(* Logix 5000 project; controller VET 1756-L62 rev 19.52; software revision 19.01; part 3 of 27 *)

        [202].S.BITS1.8   // 100-TOR-010 Atollo
        [586].S.BITS1.9   // 120-CAN-011 Conf. Cerrado
        [562].S.BITS1.9   // 110-TDC-004/2 Sobrecarga
        [318].S.BITS1.0   // 80-FIL-001 Enable
        [318].S.BITS1.1   // 80-FIL-001 Falla Resumen
        [318].S.BITS1.2   // 80-FIL-001 Conf Pos Abrir
        [318].S.BITS1.4   // 80-FIL-001 Conf Pos Cerrar
        [318].S.BITS1.26   // 80-FIL-001FLL
        [318].S.BITS1.27   // 80-FIL-001FV0
        [318].S.BITS1.28   // 80-FIL-001FATO
        [318].S.BITS1.29   // 80-FIL-001 Falla Abrir
        [318].S.BITS1.30   // 80-FIL-001 Falla Cerrar
        [318].S.BITS2.20   // 80-FIL-001 Reset Falla
        [318].S.BITS2.23   // 80-FIL-001 Test
        [318].S.BITS2.27   // 80-FIL-001 Cmd. Open
        [318].S.BITS2.30   // 80-FIL-001 OUT CLOSE
        [318].S.BITS2.31   // 80-FIL-001 OUT OPEN
        [319].S.BITS1.0   // 80-VEN-001 Enable
        [319].S.BITS1.1   // 80-VEN-001 Falla Resumen
        [319].S.BITS1.2   // 80-VEN-001 Conf. Marcha
        [319].S.BITS1.4   // 80-VEN-001 Cmd. Automatico
        [319].S.BITS1.26   // 80-VEN-001 FLL
        [319].S.BITS1.27   // 80-VEN-001 FV0
        [319].S.BITS1.28   // 80-VEN-001 FATO
        [319].S.BITS1.30   // 80-VEN-001 Falla Partida
        [319].S.BITS2.20   // 80-VEN-001 Reset Falla
        [319].S.BITS2.23   // 80-VEN-001 Test
        [319].S.BITS2.27   // 80-VEN-001 Cmd. Marcha
        [319].S.BITS2.30   // 80-VEN-001 OUT MARCHA
        [320].S.BITS1.0   // 8-VRT-638 Enable
        [320].S.BITS1.1   // 8-VRT-638 Falla Resumen
        [320].S.BITS1.2   // 8-VRT-638 Conf. Marcha
        [320].S.BITS1.4   // 8-VRT-638 Cmd. Automatico
        [320].S.BITS1.26   // 8-VRT-638 FLL
        [320].S.BITS1.27   // 8-VRT-638 FV0
        [320].S.BITS1.28   // 8-VRT-638 FATO
        [320].S.BITS1.30   // 8-VRT-638 Falla Partida
        [320].S.BITS2.20   // 8-VRT-638 Reset Falla
        [320].S.BITS2.23   // 8-VRT-638 Test
        [320].S.BITS2.27   // 8-VRT-638 Cmd. Marcha
        [320].S.BITS2.30   // 8-VRT-638 OUT MARCHA
        [322].S.BITS1.7   // 80-ENH-001 LLL
        [323].S.BITS1.0   // 8-ENF-630-2 Enable
        [323].S.BITS1.1   // 8-ENF-630-2 Falla Resumen
        [323].S.BITS1.2   // 8-ENF-630-2 Conf. Marcha
        [323].S.BITS1.4   // 8-ENF-630-2 Cmd. Automatico
        [323].S.BITS1.26   // 8-ENF-630-2 FLL
        [323].S.BITS1.27   // 8-ENF-630-2 FV0
        [323].S.BITS1.28   // 8-ENF-630-2 FATO
        [323].S.BITS1.30   // 8-ENF-630-2 Falla Partida
        [323].S.BITS2.20   // 8-ENF-630-2 Reset Falla
        [323].S.BITS2.23   // 8-ENF-630-2 Test
        [323].S.BITS2.27   // 8-ENF-630-2 Cmd. Marcha
        [323].S.BITS2.30   // 8-ENF-630-2 OUT MARCHA
        [324].S.BITS1.8   // L4-TOLV-002-B1 LL
        [235].S.BITS1.0   // 7-LRT-1189 Enable
        [325].S.BITS1.0   // 8-ENF-640-1 Enable
        [325].S.BITS1.1   // 8-ENF-640-1 Falla Resumen
        [325].S.BITS1.2   // 8-ENF-640-1 Conf. Marcha
        [325].S.BITS1.4   // 8-ENF-640-1 Cmd. Automatico
        [236].S.BITS1.0   // 100-CAN-025 Enable
        [325].S.BITS1.26   // 8-ENF-640-1 FLL
        [325].S.BITS1.27   // 8-ENF-640-1 FV0
        [325].S.BITS1.28   // 8-ENF-640-1 FATO
        [325].S.BITS1.30   // 8-ENF-640-1 Falla Partida
        [325].S.BITS2.20   // 8-ENF-640-1 Reset Falla
        [325].S.BITS2.23   // 8-ENF-640-1 Test
        [325].S.BITS2.27   // 8-ENF-640-1 Cmd. Marcha
        [325].S.BITS2.30   // 8-ENF-640-1 OUT MARCHA
        [326].S.BITS1.0   // 100-ELV-003 Enable
        [326].S.BITS1.1   // 100-ELV-003 Falla Resumen
        [326].S.BITS1.2   // 100-ELV-003 Conf. Marcha
        [326].S.BITS1.4   // 100-ELV-003 Cmd. Automatico
        [326].S.BITS1.26   // 100-ELV-003 FLL
        [326].S.BITS1.27   // 100-ELV-003 FV0
        [326].S.BITS1.28   // 100-ELV-003 FATO
        [326].S.BITS1.30   // 100-ELV-003 Falla Partida
        [326].S.BITS2.20   // 100-ELV-003 Reset Falla
        [326].S.BITS2.23   // 100-ELV-003 Test
        [326].S.BITS2.27   // 100-ELV-003 Cmd. Marcha
        [326].S.BITS2.30   // 100-ELV-003 OUT MARCHA
        [327].S.BITS1.26   // 8-ENF-640-2 FLL
        [327].S.BITS1.27   // 8-ENF-640-2 FV0
        [327].S.BITS1.28   // 8-ENF-640-2 FATO
        [328].S.BITS1.0   // 80-ESC-002/5 Enable
        [328].S.BITS1.1   // 80-ESC-002/5 Falla Resumen
        [328].S.BITS1.2   // 80-ESC-002/5 Conf. Marcha
        [328].S.BITS1.4   // 80-ESC-002/5 Cmd. Automatico
        [328].S.BITS1.26   // 80-ESC-002/5 FLL
        [328].S.BITS1.27   // 80-ESC-002/5 FV0
        [328].S.BITS1.28   // 80-ESC-002/5 FATO
        [328].S.BITS1.30   // 80-ESC-002/5 Falla Partida
        [328].S.BITS2.20   // 80-ESC-002/5 Reset Falla
        [328].S.BITS2.23   // 80-ESC-002/5 Test
        [328].S.BITS2.27   // 80-ESC-002/5 Cmd. Marcha
        [328].S.BITS2.30   // 80-ESC-002/5 OUT MARCHA
        [329].S.BITS1.0   // 80-VEN-002/5 Enable
        [329].S.BITS1.1   // 80-VEN-002/5 Falla Resumen
        [329].S.BITS1.2   // 80-VEN-002/5 Conf. Marcha
        [329].S.BITS1.4   // 80-VEN-002/5 Cmd. Automatico
        [329].S.BITS1.26   // 80-VEN-002/5 FLL
        [329].S.BITS1.27   // 80-VEN-002/5 FV0
        [329].S.BITS1.28   // 80-VEN-002/5 FATO
        [329].S.BITS1.30   // 80-VEN-002/5 Falla Partida
        [329].S.BITS2.20   // 80-VEN-002/5 Reset Falla
        [329].S.BITS2.23   // 80-VEN-002/5 Test
        [329].S.BITS2.27   // 80-VEN-002/5 Cmd. Marcha
        [329].S.BITS2.30   // 80-VEN-002/5 OUT MARCHA
        [331].S.BITS1.0   // 80-TOR-004/5 Enable
        [331].S.BITS1.1   // 80-TOR-004/5 Falla Resumen
        [331].S.BITS1.2   // 80-TOR-004/5 Conf. Marcha
        [331].S.BITS1.4   // 80-TOR-004/5 Cmd. Automatico
        [331].S.BITS1.26   // 80-TOR-004/5 FLL
        [331].S.BITS1.27   // 80-TOR-004/5 FV0
        [331].S.BITS1.28   // 80-TOR-004/5 FATO
        [331].S.BITS1.30   // 80-TOR-004/5 Falla Partida
        [331].S.BITS2.20   // 80-TOR-004/5 Reset Falla
        [331].S.BITS2.23   // 80-TOR-004/5 Test
        [331].S.BITS2.27   // 80-TOR-004/5 Cmd. Marcha
        [331].S.BITS2.30   // 80-TOR-004/5 OUT MARCHA
        [332].S.BITS1.0   // 8-VEN-647 Enable
        [332].S.BITS1.1   // 8-VEN-647 Falla Resumen
        [332].S.BITS1.2   // 8-VEN-647 Conf. Marcha
        [332].S.BITS1.4   // 8-VEN-647 Cmd. Automatico
        [332].S.BITS1.26   // 8-VEN-647 FLL
        [332].S.BITS1.27   // 8-VEN-647 FV0
        [332].S.BITS1.28   // 8-VEN-647 FATO
        [332].S.BITS1.30   // 8-VEN-647 Falla Partida
        [332].S.BITS2.20   // 8-VEN-647 Reset Falla
        [332].S.BITS2.23   // 8-VEN-647 Test
        [332].S.BITS2.27   // 8-VEN-647 Cmd. Marcha
        [332].S.BITS2.30   // 8-VEN-647 OUT MARCHA
        [333].S.BITS1.0   // 8-ENF-640-2 Enable
        [333].S.BITS1.1   // 8-ENF-640-2 Falla Resumen
        [333].S.BITS1.2   // 8-ENF-640-2 Conf. Marcha
        [333].S.BITS1.4   // 8-ENF-640-2 Cmd. Automatico
        [333].S.BITS1.26   // 8-ENF-640-2 FLL
        [333].S.BITS1.27   // 8-ENF-640-2 FV0
        [333].S.BITS1.28   // 8-ENF-640-2 FATO
        [333].S.BITS1.30   // 8-ENF-640-2 Falla Partida
        [333].S.BITS2.20   // 8-ENF-640-2 Reset Falla
        [333].S.BITS2.23   // 8-ENF-640-2 Test
        [333].S.BITS2.27   // 8-ENF-640-2 Cmd. Marcha
        [333].S.BITS2.30   // 8-ENF-640-2 OUT MARCHA
        [564].S.BITS1.9   // 110-ELV-001/2 Sobrecarga
        [236].S.BITS2.30   // 100-CAN-025 OUT CLOSE
        [355].S.BITS1.10   // 110-CAN-003 Conf. Abierto
        [587].S.BITS1.9   // 120-CAN-012 Conf. Cerrado
        [239].S.BITS2.31   // 7-CON-1192 OUT OPEN
        [242].S.BITS2.31   // 7-CON-1195 OUT OPEN
        [280].S.BITS1.8   // 100-DOS-100-M10 Atollo
        [335].S.BITS1.0   // 8-ROS-654 Enable
        [335].S.BITS1.1   // 8-ROS-654 Falla Resumen
        [335].S.BITS1.2   // 8-ROS-654 Conf. Marcha
        [335].S.BITS1.4   // 8-ROS-654 Cmd. Automatico
        [335].S.BITS1.26   // 8-ROS-654 FLL
        [335].S.BITS1.27   // 8-ROS-654 FV0
        [335].S.BITS1.28   // 8-ROS-654 FATO
        [335].S.BITS1.30   // 8-ROS-654 Falla Partida
        [335].S.BITS2.20   // 8-ROS-654 Reset Falla
        [335].S.BITS2.23   // 8-ROS-654 Test
        [335].S.BITS2.27   // 8-ROS-654 Cmd. Marcha
        [335].S.BITS2.30   // 8-ROS-654 OUT MARCHA
        [336].S.BITS1.0   // 8-ELV-656 Enable
        [336].S.BITS1.1   // 8-ELV-656 Falla Resumen
        [336].S.BITS1.2   // 8-ELV-656 Conf. Marcha
        [336].S.BITS1.4   // 8-ELV-656 Cmd. Automatico
        [336].S.BITS1.26   // 8-ELV-656 FLL
        [336].S.BITS1.27   // 8-ELV-656 FV0
        [336].S.BITS1.28   // 8-ELV-656 FATO
        [336].S.BITS1.30   // 8-ELV-656 Falla Partida
        [336].S.BITS2.20   // 8-ELV-656 Reset Falla
        [336].S.BITS2.23   // 8-ELV-656 Test
        [336].S.BITS2.27   // 8-ELV-656 Cmd. Marcha
        [336].S.BITS2.30   // 8-ELV-656 OUT MARCHA
        [565].S.BITS1.9   // 120-TDC-001/2 Sobrecarga
        [244].S.BITS2.31   // 100-TOR-020 OUT MARCHA
        [356].S.BITS1.10   // 110-CAN-004 Conf. Abierto
        [588].S.BITS1.9   // 120-CAN-013 Conf. Cerrado
        [246].S.BITS2.31   // 100-TOR-019 OUT MARCHA
        [248].S.BITS2.31   // 100-TOR-018 OUT MARCHA
        [282].S.BITS1.8   // 100-DOS-100-M11 Atollo
        [338].S.BITS1.0   // 8-RED-660 Enable
        [338].S.BITS1.1   // 8-RED-660 Falla Resumen
        [338].S.BITS1.2   // 8-RED-660 Conf. Marcha
        [338].S.BITS1.4   // 8-RED-660 Cmd. Automatico
        [338].S.BITS1.7   // TOLV-008 LLL
        [338].S.BITS1.8   // TOLV-008 LL
        [338].S.BITS1.9   // TOLV-008 LM
        [338].S.BITS1.10   // TOLV-008 LH
        [338].S.BITS1.26   // 8-RED-660 FLL
        [338].S.BITS1.27   // 8-RED-660 FV0
        [338].S.BITS1.28   // 8-RED-660 FATO
        [338].S.BITS1.30   // 8-RED-660 Falla Partida
        [338].S.BITS2.20   // 8-RED-660 Reset Falla
        [338].S.BITS2.23   // 8-RED-660 Test
        [338].S.BITS2.27   // 8-RED-660 Cmd. Marcha
        [338].S.BITS2.30   // 8-RED-660 OUT MARCHA
        [339].S.BITS1.0   // 8-ELV-662 Enable
        [339].S.BITS1.1   // 8-ELV-662 Falla Resumen
        [339].S.BITS1.2   // 8-ELV-662 Conf. Marcha
        [339].S.BITS1.4   // 8-ELV-662 Cmd. Automatico
        [339].S.BITS1.26   // 8-ELV-662 FLL
        [339].S.BITS1.27   // 8-ELV-662 FV0
        [339].S.BITS1.28   // 8-ELV-662 FATO
        [339].S.BITS1.29   // CV-ENF-L1 Falla Abrir
        [339].S.BITS2.20   // 8-ELV-662 Reset Falla
        [339].S.BITS2.23   // 8-ELV-662 Test
        [339].S.BITS2.31   // CV-ENF-L1 OUT OPEN
        [340].S.BITS1.0   // 8-ZRD-664 Enable
        [340].S.BITS1.1   // 8-ZRD-664 Falla Resumen
        [340].S.BITS1.2   // 8-ZRD-664 Conf. Marcha
        [340].S.BITS1.4   // 8-ZRD-664 Cmd. Automatico
        [340].S.BITS1.7   // 80-TOL-004/6 LLL
        [340].S.BITS1.8   // 80-TOL-004/6 LL
        [340].S.BITS1.9   // 80-TOL-004/6 LM
        [340].S.BITS1.10   // 80-TOL-004/6 LH
        [340].S.BITS1.26   // 8-ZRD-664 FLL
        [340].S.BITS1.27   // 8-ZRD-664 FV0
        [340].S.BITS1.28   // 8-ZRD-664 FATO
        [340].S.BITS1.30   // 8-ZRD-664 Falla Partida
        [340].S.BITS2.20   // 8-ZRD-664 Reset Falla
        [340].S.BITS2.23   // 8-ZRD-664 Test
        [340].S.BITS2.27   // 8-ZRD-664 Cmd. Marcha
        [340].S.BITS2.30   // 8-ZRD-664 OUT MARCHA
        [341].S.BITS1.0   // 8-RED-666 Enable
        [341].S.BITS1.1   // 8-RED-666 Falla Resumen
        [341].S.BITS1.2   // 8-RED-666 Conf. Marcha
        [341].S.BITS1.4   // 8-RED-666 Cmd. Automatico
        [341].S.BITS1.26   // 8-RED-666 FLL
        [341].S.BITS1.27   // 8-RED-666 FV0
        [341].S.BITS1.28   // 8-RED-666 FATO
        [341].S.BITS1.30   // 8-RED-666 Falla Partida
        [341].S.BITS2.20   // 8-RED-666 Reset Falla
        [341].S.BITS2.23   // 8-RED-666 Test
        [341].S.BITS2.27   // 8-RED-666 Cmd. Marcha
        [341].S.BITS2.30   // 8-RED-666 OUT MARCHA
        [342].S.BITS1.0   // 8-CON-664b Enable
        [342].S.BITS1.1   // 8-CON-664b Falla Resumen
        [342].S.BITS1.4   // 8-CON-664b Conf Pos Cerrar
        [342].S.BITS1.26   // 110-TDC-001 FLL
        [342].S.BITS1.27   // 110-TDC-001 FV0
        [342].S.BITS1.28   // 110-TDC-001 FATO
        [342].S.BITS1.30   // 8-CON-664b Falla Cerrar
        [342].S.BITS2.20   // 8-CON-664b Reset Falla
        [342].S.BITS2.23   // 8-CON-664b Test
        [342].S.BITS2.27   // 8-CON-664b Cmd. Open
        [342].S.BITS2.30   // 8-CON-664b OUT CLOSE
        [343].S.BITS1.0   // COM-VIR-1 Enable
        [343].S.BITS1.1   // COM-VIR-1 Falla Resumen
        [343].S.BITS1.2   // COM-VIR-1 Conf Pos Abrir
        [343].S.BITS1.4   // COM-VIR-1 Conf Pos Cerrar
        [343].S.BITS1.29   // COM-VIR-1 Falla Abrir
        [343].S.BITS1.30   // COM-VIR-1 Falla Cerrar
        [343].S.BITS2.20   // COM-VIR-1 Reset Falla
        [343].S.BITS2.23   // COM-VIR-1 Test
        [343].S.BITS2.27   // COM-VIR-1 Cmd. Open
        [343].S.BITS2.30   // COM-VIR-1 OUT CLOSE
        [343].S.BITS2.31   // COM-VIR-1 OUT OPEN
        [337].S.BITS1.8   // 110-VEN-003 Atollo
        [357].S.BITS1.10   // 110-CAN-005 Conf. Abierto
        [589].S.BITS1.9   // 120-CAN-014 Conf. Cerrado
        [169].S.BITS1.10   // 100-VEN-002 Velocidad Cero
        [344].S.BITS1.26   // 80-EXP-002/6 FLL
        [344].S.BITS1.27   // 80-EXP-002/6 FV0
        [344].S.BITS1.28   // 80-EXP-002/6 FATO
        [116].S.BITS1.10   // 100-ELV-001 Velocidad Cero
        [590].S.BITS1.9   // 120-CAN-015 Conf. Cerrado
        [205].S.BITS1.8   // 100-TOR-036 Atollo
        [344].S.BITS2.27   // 110-LMG-001-01 Cmd. Open
        [571].S.BITS1.9   // 110-TDC-003/3 Sobrecarga
        [345].S.BITS1.0   // 80-DES-002/6 Enable
        [345].S.BITS1.1   // 80-DES-002/6 Falla Resumen
        [345].S.BITS1.2   // 80-DES-002/6 Conf. Marcha
        [345].S.BITS1.4   // 80-DES-002/6 Cmd. Automatico
        [345].S.BITS1.26   // 80-DES-002/6 FLL
        [345].S.BITS1.27   // 80-DES-002/6 FV0
        [345].S.BITS1.28   // 80-DES-002/6 FATO
        [345].S.BITS1.30   // 80-DES-002/6 Falla Partida
        [345].S.BITS2.20   // 80-DES-002/6 Reset Falla
        [345].S.BITS2.23   // 80-DES-002/6 Test
        [345].S.BITS2.27   // 80-DES-002/6 Cmd. Marcha
        [345].S.BITS2.30   // 80-DES-002/6 OUT MARCHA
        [346].S.BITS1.0   // 110-LMG-002 Enable
        [346].S.BITS1.1   // 110-LMG-002 Falla Resumen
        [592].S.BITS1.9   // 120-CAN-027 Conf. Cerrado
        [172].S.BITS1.10   // 100-TOR-001 Velocidad Cero
        [346].S.BITS1.26   // 80-PLT-001/6 FLL
        [346].S.BITS1.27   // 80-PLT-001/6 FV0
        [346].S.BITS1.28   // 80-PLT-001/6 FATO
        [122].S.BITS1.10   // 100-TDP-001 Velocidad Cero
        [346].S.BITS2.20   // 110-LMG-002 Reset Falla
        [346].S.BITS2.23   // 110-LMG-002 Test
        [593].S.BITS1.9   // 120-CAN-028 Conf. Cerrado
        [572].S.BITS1.9   // 110-TDC-004/3 Sobrecarga
        [347].S.BITS1.0   // 80-CAE-001/6 Enable
        [347].S.BITS1.1   // 80-CAE-001/6 Falla Resumen
        [347].S.BITS1.2   // 80-CAE-001/6 Conf. Marcha
        [347].S.BITS1.4   // 80-CAE-001/6 Cmd. Automatico
        [347].S.BITS1.26   // 80-CAE-001/6 FLL
        [347].S.BITS1.27   // 80-CAE-001/6 FV0
        [347].S.BITS1.28   // 80-CAE-001/6 FATO
        [347].S.BITS1.30   // 80-CAE-001/6 Falla Partida
        [347].S.BITS2.20   // 80-CAE-001/6 Reset Falla
        [347].S.BITS2.23   // 80-CAE-001/6 Test
        [347].S.BITS2.27   // 80-CAE-001/6 Cmd. Marcha
        [347].S.BITS2.30   // 80-CAE-001/6 OUT MARCHA
        [348].S.BITS1.0   // 8-ROS-710 Enable
        [348].S.BITS1.1   // 8-ROS-710 Falla Resumen
        [348].S.BITS1.2   // 8-ROS-710 Conf. Marcha
        [348].S.BITS1.4   // 8-ROS-710 Cmd. Automatico
        [348].S.BITS1.7   // TOL_VIR_DESP-01 LLL
        [348].S.BITS1.8   // 110-TOL-002 LL
        [348].S.BITS1.9   // 110-TOL-002 LM
        [348].S.BITS1.10   // 110-TOL-002 LH
        [348].S.BITS1.26   // 8-ROS-710 FLL
        [348].S.BITS1.27   // 8-ROS-710 FV0
        [348].S.BITS1.28   // 8-ROS-710 FATO
        [348].S.BITS1.30   // 8-ROS-710 Falla Partida
        [348].S.BITS2.20   // 8-ROS-710 Reset Falla
        [348].S.BITS2.23   // 8-ROS-710 Test
        [348].S.BITS2.27   // 8-ROS-710 Cmd. Marcha
        [348].S.BITS2.30   // 8-ROS-710 OUT MARCHA
        [349].S.BITS1.0   // 110-LRT-001 Enable
        [349].S.BITS1.1   // 110-LRT-001 Falla Resumen
        [349].S.BITS1.2   // 110-LRT-001 Conf. Marcha
        [349].S.BITS1.4   // 110-LRT-001 Cmd. Automatico
        [349].S.BITS1.29   // COM-VIR-DESP-01 Falla Abrir
        [349].S.BITS1.30   // 110-LRT-001 Falla Partida
        [349].S.BITS2.20   // 110-LRT-001 Reset Falla
        [349].S.BITS2.23   // 110-LRT-001 Test
        [349].S.BITS2.27   // 110-LRT-001 Cmd. Marcha
        [349].S.BITS2.30   // 110-LRT-001 OUT MARCHA
        [349].S.BITS2.31   // 110-LRT-001 OUT MARCHA
        [350].S.BITS1.7   // TOL_VIR_DESP-01 LLL
        [350].S.BITS1.8   // 110-TOL-003 LL
        [350].S.BITS1.9   // 110-TOL-003 LM
        [350].S.BITS1.10   // 110-TOL-003 LH
        [350].S.BITS2.11   // RED-063-00 Enc Ext
        [350].S.BITS2.31   // RED-063-00 Out
        [351].S.BITS1.0   // 8-ACO-716 Enable
        [351].S.BITS1.1   // 8-ACO-716 Falla Resumen
        [351].S.BITS1.2   // 8-ACO-716 Conf. Marcha
        [351].S.BITS1.4   // 8-ACO-716 Cmd. Automatico
        [351].S.BITS1.29   // COM-VIR-DESP-01 Falla Abrir
        [351].S.BITS1.30   // 8-ACO-716 Falla Partida
        [351].S.BITS2.20   // 8-ACO-716 Reset Falla
        [351].S.BITS2.23   // 8-ACO-716 Test
        [351].S.BITS2.27   // 8-ACO-716 Cmd. Marcha
        [351].S.BITS2.30   // 8-ACO-716 OUT MARCHA
        [351].S.BITS2.31   // 110-TOR-005 OUT MARCHA
        [573].S.BITS1.9   // 110-TDC-005/3 Sobrecarga
        [250].S.BITS2.31   // 100-TOR-017 OUT MARCHA
        [358].S.BITS1.10   // 8-ENF-730 LH
        [352].S.BITS1.7   // 80-ENH-001 LLL
        [352].S.BITS1.10   // 110-TDC-002 Velocidad Cero
        [594].S.BITS1.9   // 120-CAN-029 Conf. Cerrado
        [252].S.BITS2.31   // 100-TOR-016 OUT MARCHA
        [288].S.BITS2.31   // 100-DOS-001-C OUT OPEN
        [284].S.BITS1.8   // 100-DOS-100-M12 Atollo
        [353].S.BITS1.0   // 8-PLT-722 Enable
        [353].S.BITS1.1   // 8-PLT-722 Falla Resumen
        [595].S.BITS1.9   // 120-CAN-030 Conf. Cerrado
        [353].S.BITS1.4   // 8-PLT-722 Cmd. Automatico
        [353].S.BITS1.26   // 8-PLT-722 FLL
        [353].S.BITS1.27   // 8-PLT-722 FV0
        [353].S.BITS1.28   // 8-PLT-722 FATO
        [353].S.BITS1.30   // 8-PLT-722 Falla Partida
        [353].S.BITS2.20   // 8-PLT-722 Reset Falla
        [353].S.BITS2.23   // 8-PLT-722 Test
        [353].S.BITS2.27   // 8-PLT-722 Cmd. Marcha
        [353].S.BITS2.30   // 8-PLT-722 OUT MARCHA
        [289].S.BITS1.9   // 100-TDP-003 Sobrecarga
        [546].S.BITS1.8   // 110-ELV-002/3 Atollo
        [574].S.BITS1.9   // 110-ELV-001/3 Sobrecarga
        [354].S.BITS1.26   // L4-VAPOR FLL
        [354].S.BITS1.27   // L4-VAPOR FV0
        [354].S.BITS1.28   // L4-VAPOR FATO
        [289].S.BITS2.31   // 100-TDP-003 OUT MARCHA
        [548].S.BITS1.8   // 110-TOR-004/3 Atollo
        [551].S.BITS1.8   // 110-TDC-003/1 Atollo
        [450].S.BITS1.8   // 9-BIN-712 LL
        [355].S.BITS1.0   // 110-CAN-003 Enable
        [355].S.BITS1.1   // 110-CAN-003 Falla Resumen
        [596].S.BITS1.9   // 120-CAN-031 Conf. Cerrado
        [355].S.BITS1.4   // 110-CAN-003 Conf Pos Cerrar
        [355].S.BITS1.26   // 80-CIC-001/6 FLL
        [355].S.BITS1.27   // 80-CIC-001/6 FV0
        [355].S.BITS1.28   // 80-CIC-001/6 FATO
        [355].S.BITS1.30   // 110-CAN-003 Falla Cerrar
        [355].S.BITS2.20   // 110-CAN-003 Reset Falla
        [355].S.BITS2.23   // 110-CAN-003 Test
        [355].S.BITS2.27   // 110-CAN-003 Cmd. Open
        [355].S.BITS2.30   // 110-CAN-003 OUT CLOSE
        [356].S.BITS1.0   // 8-VRT-729 Enable
        [356].S.BITS1.1   // 8-VRT-729 Falla Resumen
        [602].S.BITS1.9   // 120-CAN-039 Conf. Cerrado
        [356].S.BITS1.4   // 8-VRT-729 Cmd. Automatico
        [356].S.BITS1.26   // 8-VRT-729 FLL
        [356].S.BITS1.27   // 8-VRT-729 FV0
        [356].S.BITS1.28   // 8-VRT-729 FATO
        [356].S.BITS1.30   // 8-VRT-729 Falla Partida
        [356].S.BITS2.20   // 8-VRT-729 Reset Falla
        [356].S.BITS2.23   // 8-VRT-729 Test
        [356].S.BITS2.27   // 8-VRT-729 Cmd. Marcha
        [356].S.BITS2.30   // 8-VRT-729 OUT MARCHA
        [357].S.BITS1.0   // 8-ENF-730-1 Enable
        [357].S.BITS1.1   // 8-ENF-730-1 Falla Resumen
        [603].S.BITS1.9   // 120-CAN-040 Conf. Cerrado
        [357].S.BITS1.4   // 8-ENF-730-1 Cmd. Automatico
        [357].S.BITS1.26   // 8-ENF-730-1 FLL
        [357].S.BITS1.27   // 8-ENF-730-1 FV0
        [357].S.BITS1.28   // 8-ENF-730-1 FATO
        [357].S.BITS2.20   // 8-ENF-730-1 Reset Falla
        [357].S.BITS2.23   // 8-ENF-730-1 Test
        [358].S.BITS1.0   // 110-CAN-006 Enable
        [358].S.BITS1.1   // 110-CAN-006 Falla Resumen
        [604].S.BITS1.9   // 120-CAN-041 Conf. Cerrado
        [358].S.BITS1.4   // 110-CAN-006 Conf Pos Cerrar
        [358].S.BITS1.26   // 80-ESC-002/6 FLL
        [358].S.BITS1.27   // 80-ESC-002/6 FV0
        [358].S.BITS1.28   // 80-ESC-002/6 FATO
        [358].S.BITS1.30   // 110-CAN-006 Falla Cerrar
        [358].S.BITS2.20   // 110-CAN-006 Reset Falla
        [358].S.BITS2.23   // 110-CAN-006 Test
        [358].S.BITS2.27   // 110-CAN-006 Cmd. Open
        [358].S.BITS2.30   // 110-CAN-006 OUT CLOSE
        [359].S.BITS1.0   // 8-ENF-730-2 Enable
        [359].S.BITS1.1   // 8-ENF-730-2 Falla Resumen
        [359].S.BITS1.2   // 8-ENF-730-2 Conf. Marcha
        [359].S.BITS1.4   // 8-ENF-730-2 Cmd. Automatico
        [359].S.BITS1.26   // 8-ENF-730-2 FLL
        [359].S.BITS1.27   // 8-ENF-730-2 FV0
        [359].S.BITS1.28   // 8-ENF-730-2 FATO
        [359].S.BITS1.30   // 8-ENF-730-2 Falla Partida
        [359].S.BITS2.20   // 8-ENF-730-2 Reset Falla
        [359].S.BITS2.23   // 8-ENF-730-2 Test
        [359].S.BITS2.27   // 8-ENF-730-2 Cmd. Marcha
        [359].S.BITS2.30   // 8-ENF-730-2 OUT MARCHA
        [360].S.BITS1.8   // TOL-VIR-2 LL
        [360].S.BITS1.9   // TOL-VIR-2 LM
        [360].S.BITS1.10   // TOL-VIR-2 LH
        [361].S.BITS1.0   // 80-TOR-004/6 Enable
        [361].S.BITS1.1   // 80-TOR-004/6 Falla Resumen
        [361].S.BITS1.2   // 80-TOR-004/6 Conf. Marcha
        [361].S.BITS1.4   // 80-TOR-004/6 Cmd. Automatico
        [361].S.BITS1.26   // 80-TOR-004/6 FLL
        [361].S.BITS1.27   // 80-TOR-004/6 FV0
        [361].S.BITS1.28   // 80-TOR-004/6 FATO
        [361].S.BITS1.29   // COM-VIR-2 Falla Abrir
        [361].S.BITS1.30   // 80-TOR-004/6 Falla Partida
        [361].S.BITS2.20   // 80-TOR-004/6 Reset Falla
        [361].S.BITS2.23   // 80-TOR-004/6 Test
        [361].S.BITS2.27   // 80-TOR-004/6 Cmd. Marcha
        [361].S.BITS2.30   // 80-TOR-004/6 OUT MARCHA
        [361].S.BITS2.31   // COM-VIR-2 OUT OPEN
        [362].S.BITS1.0   // 8-VRT-736 Enable
        [362].S.BITS1.1   // 8-VRT-736 Falla Resumen
        [362].S.BITS1.2   // 8-VRT-736 Conf. Marcha
        [362].S.BITS1.4   // 8-VRT-736 Cmd. Automatico
        [362].S.BITS1.26   // 8-VRT-736 FLL
        [362].S.BITS1.27   // 8-VRT-736 FV0
        [362].S.BITS1.28   // 8-VRT-736 FATO
        [362].S.BITS1.30   // 8-VRT-736 Falla Partida
        [362].S.BITS2.20   // 8-VRT-736 Reset Falla
        [362].S.BITS2.23   // 8-VRT-736 Test
        [362].S.BITS2.27   // 8-VRT-736 Cmd. Marcha
        [362].S.BITS2.30   // 8-VRT-736 OUT MARCHA
        [342].S.BITS1.8   // 110-TDC-001 Atollo
        [382].S.BITS1.9   // 110-ENF-001/1-4 Sobrecarga
        [605].S.BITS1.9   // 120-CAN-042 Conf. Cerrado
        [178].S.BITS1.10   // 7-DOS-1170-03 LH
        [363].S.BITS1.26   // 80-ELV-002/6 FLL
        [363].S.BITS1.27   // 80-ELV-002/6 FV0
        [363].S.BITS1.28   // 80-ELV-002/6 FATO
        [363].S.BITS1.30   // 110-CAN-008/1 Falla Cerrar
        [606].S.BITS1.9   // 120-CAN-043 Conf. Cerrado
        [208].S.BITS1.8   // 100-TOR-012 Atollo
        [363].S.BITS2.27   // 110-CAN-008/1 Cmd. Open
        [363].S.BITS2.30   // 110-CAN-008/1 OUT CLOSE
        [349].S.BITS1.8   // 8-TOL-712 LL
        [384].S.BITS1.9   // 110-ENF-001/1-1 Sobrecarga
        [607].S.BITS1.9   // 120-CAN-044 Conf. Cerrado
        [181].S.BITS1.10   // 100-TOR-004 Velocidad Cero
        [211].S.BITS1.8   // 100-TOR-013 Atollo
        [131].S.BITS1.10   // 100-TDC-001 Velocidad Cero
        [608].S.BITS1.9   // 120-CAN-045 Conf. Cerrado
        [214].S.BITS1.8   // 7-ETQ-1179a LL
        [612].S.BITS1.9   // 120-CAN-055 Conf. Cerrado
        [575].S.BITS1.9   // 120-TDC-001/3 Sobrecarga
        [366].S.BITS1.0   // 8-VRT-739 Enable
        [366].S.BITS1.1   // 8-VRT-739 Falla Resumen
        [366].S.BITS1.2   // 8-VRT-739 Conf. Marcha
        [366].S.BITS1.4   // 8-VRT-739 Cmd. Automatico
        [366].S.BITS1.26   // 8-VRT-739 FLL
        [366].S.BITS1.27   // 8-VRT-739 FV0
        [366].S.BITS1.28   // 8-VRT-739 FATO
        [366].S.BITS1.30   // 8-VRT-739 Falla Partida
        [366].S.BITS2.20   // 8-VRT-739 Reset Falla
        [366].S.BITS2.23   // 8-VRT-739 Test
        [366].S.BITS2.27   // 8-VRT-739 Cmd. Marcha
        [366].S.BITS2.30   // 8-VRT-739 OUT MARCHA
        [367].S.BITS1.0   // 8-ENF-740-1 Enable
        [367].S.BITS1.1   // 8-ENF-740-1 Falla Resumen
        [367].S.BITS1.2   // 8-ENF-740-1 Conf. Marcha
        [367].S.BITS1.4   // 8-ENF-740-1 Cmd. Automatico
        [367].S.BITS1.26   // 8-ENF-740-1 FLL
        [367].S.BITS1.27   // 8-ENF-740-1 FV0
        [367].S.BITS1.28   // 8-ENF-740-1 FATO
        [367].S.BITS1.30   // 8-ENF-740-1 Falla Partida
        [367].S.BITS2.20   // 8-ENF-740-1 Reset Falla
        [367].S.BITS2.23   // 8-ENF-740-1 Test
        [367].S.BITS2.27   // 8-ENF-740-1 Cmd. Marcha
        [367].S.BITS2.30   // 8-ENF-740-1 OUT MARCHA
        [368].S.BITS1.7   // TOLV-007 LLL
        [369].S.BITS1.2   // 8-ENF-740-2 Conf. Marcha
        [369].S.BITS1.8   // 110-TOL-005/1 LL
        [369].S.BITS1.9   // 110-TOL-005/1 LM
        [369].S.BITS1.10   // 110-TOL-005/1 LH
        [369].S.BITS1.29   // CV-ENF-L2 Falla Abrir
        [369].S.BITS2.31   // CV-ENF-L2 OUT OPEN
        [678].S.BITS1.29   // 120-CAN-067 Falla Abrir
        [297].S.BITS2.31   // 100-TOL-003-1 OUT OPEN
        [389].S.BITS1.9   // 110-VAL-001/1-1 Sobrecarga
        [613].S.BITS1.9   // 120-CAN-056 Conf. Cerrado
        [302].S.BITS2.31   // 100-BCE-003 OUT MARCHA
        [304].S.BITS2.31   // 100-BCE-005 OUT MARCHA
        [292].S.BITS1.9   // 100-TDP-004 Sobrecarga
        [371].S.BITS1.0   // 90-HAR-001-C Enable
        [371].S.BITS1.1   // 90-HAR-001-C Falla Resumen
        [371].S.BITS1.2   // 90-HAR-001-C Conf Pos Abrir
        [371].S.BITS1.4   // 90-HAR-001-C Conf Pos Cerrar
        [371].S.BITS1.26   // L3-ROS-014 FLL
        [371].S.BITS1.27   // L3-ROS-014 FV0
        [371].S.BITS1.28   // L3-ROS-014 FATO
        [371].S.BITS1.29   // 90-HAR-001-C Falla Abrir
        [371].S.BITS1.30   // 90-HAR-001-C Falla Cerrar
        [371].S.BITS2.20   // 90-HAR-001-C Reset Falla
        [371].S.BITS2.23   // 90-HAR-001-C Test
        [371].S.BITS2.27   // 90-HAR-001-C Cmd. Open
        [371].S.BITS2.30   // 90-HAR-001-C OUT CLOSE
        [371].S.BITS2.31   // 90-HAR-001-C OUT OPEN
        [678].S.BITS2.20   // 120-CAN-067 Reset Falla
        [308].S.BITS2.31   // 100-BCE-002 OUT MARCHA
        [390].S.BITS1.9   // 110-VEN-001/1-1 Sobrecarga
        [614].S.BITS1.9   // 120-CAN-057 Conf. Cerrado
        [312].S.BITS2.31   // 8-BIF-624 Out Derecha
        [323].S.BITS2.31   // 100-VIB-001 OUT MARCHA
        [293].S.BITS1.9   // 100-ELV-002 Sobrecarga
        [351].S.BITS1.8   // 110-TOR-005 Atollo
        [391].S.BITS1.9   // 110-ENF-001/1-5 Sobrecarga
        [615].S.BITS1.9   // 120-CAN-058 Conf. Cerrado
        [184].S.BITS1.10   // 7-DOS-1170-06 LH
        [217].S.BITS1.8   // 7-ETQ-1179b LL
        [134].S.BITS1.10   // 7-TOL-1137 LH
        [616].S.BITS1.9   // 120-CAN-059 Conf. Cerrado
        [218].S.BITS1.8   // 100-TOR-038 Atollo
        [617].S.BITS1.9   // 120-CAN-060 Conf. Cerrado
        [680].S.BITS1.29   // 120-CAN-068 Falla Abrir
        [680].S.BITS2.20   // 120-CAN-068 Reset Falla
        [325].S.BITS2.31   // 100-TDC-007 OUT MARCHA
        [402].S.BITS1.9   // 110-ENF-002/1-4 Sobrecarga
        [618].S.BITS1.9   // 120-CAN-061 Conf. Cerrado
        [326].S.BITS2.31   // 100-ELV-003 OUT MARCHA
        [332].S.BITS2.31   // 110-FIL-001 OUT MARCHA
        [294].S.BITS1.9   // 100-TDP-005 Sobrecarga
        [352].S.BITS1.8   // 110-TDC-002 Atollo
        [404].S.BITS1.9   // 110-ENF-002/1-1 Sobrecarga
        [375].S.BITS1.2   // 8-ENF-740-2 Conf. Marcha
        [187].S.BITS1.10   // 100-TOR-006 Velocidad Cero
        [375].S.BITS1.29   // 90-HAR-002-C Falla Abrir
        [409].S.BITS1.9   // 110-VAL-002/1-1 Sobrecarga
        [622].S.BITS1.9   // 120-CAN-017 Conf. Cerrado
        [220].S.BITS1.8   // 7-ETQ-1179c LL
        [334].S.BITS2.31   // 110-FIL-002 OUT MARCHA
        [336].S.BITS2.31   // 110-FIL-003 OUT MARCHA
        [375].S.BITS2.31   // 110-CAE-001/1 OUT MARCHA
        [682].S.BITS1.29   // 120-CAN-069 Falla Abrir
        [337].S.BITS2.31   // 110-VEN-003 OUT MARCHA
        [410].S.BITS1.9   // 110-VEN-002/1-1 Sobrecarga
        [624].S.BITS1.9   // 120-CAN-018 Conf. Cerrado
        [342].S.BITS2.31   // 8-CON-664b OUT OPEN
        [352].S.BITS2.31   // 110-TDC-002 OUT MARCHA
        [302].S.BITS1.9   // 100-BCE-003 Sobrecarga
        [556].S.BITS1.8   // 120-HAR-001 Atollo
        [411].S.BITS1.9   // 110-ENF-002/1-5 Sobrecarga
        [626].S.BITS1.9   // 120-CAN-019 Conf. Cerrado
        [193].S.BITS1.10   // 100-TOR-007 Velocidad Cero
        [377].S.BITS1.26   // 8-ROS-754 FLL
        [377].S.BITS1.27   // 8-ROS-754 FV0
        [377].S.BITS1.28   // 8-ROS-754 FATO
        [142].S.BITS1.10   // 100-TDC-003 Velocidad Cero
        [628].S.BITS1.9   // 120-CAN-020 Conf. Cerrado
        [223].S.BITS1.8   // 7-TOL-1180 LL
        [630].S.BITS1.9   // 120-CAN-021 Conf. Cerrado
        [682].S.BITS2.20   // 120-CAN-069 Reset Falla
        [378].S.BITS1.0   // 8-ELV-756 Enable
        [378].S.BITS1.1   // 8-ELV-756 Falla Resumen
        [378].S.BITS1.2   // 8-ELV-756 Conf. Marcha
        [378].S.BITS1.4   // 8-ELV-756 Cmd. Automatico
        [378].S.BITS1.8   // L4-TOLV-CIC-01 LL
        [378].S.BITS1.9   // L4-TOLV-CIC-01 LM
        [378].S.BITS1.10   // L4-TOLV-CIC-01 LH
        [378].S.BITS1.26   // 8-ELV-756 FLL
        [378].S.BITS1.27   // 8-ELV-756 FV0
        [378].S.BITS1.28   // 8-ELV-756 FATO
        [378].S.BITS1.30   // 8-ELV-756 Falla Partida
        [378].S.BITS2.20   // 8-ELV-756 Reset Falla
        [378].S.BITS2.23   // 8-ELV-756 Test
        [378].S.BITS2.27   // 8-ELV-756 Cmd. Marcha
        [378].S.BITS2.30   // 8-ELV-756 OUT MARCHA
        [379].S.BITS1.0   // 8-RED-758 Enable
        [379].S.BITS1.1   // 8-RED-758 Falla Resumen
        [379].S.BITS1.2   // 8-RED-758 Conf. Marcha
        [379].S.BITS1.4   // 8-RED-758 Cmd. Automatico
        [379].S.BITS1.8   // L4-TOLV-CIC-02 LL
        [379].S.BITS1.9   // L4-TOLV-CIC-02 LM
        [379].S.BITS1.10   // L4-TOLV-CIC-02 LH
        [379].S.BITS1.29   // 90-CAN-001 Falla Abrir
        [379].S.BITS1.30   // 8-RED-758 Falla Partida
        [379].S.BITS2.20   // 8-RED-758 Reset Falla
        [379].S.BITS2.23   // 8-RED-758 Test
        [379].S.BITS2.30   // 8-RED-758 OUT MARCHA
        [379].S.BITS2.31   // 90-CAN-001 OUT OPEN
        [380].S.BITS1.0   // 8-RED-760 Enable
        [380].S.BITS1.1   // 8-RED-760 Falla Resumen
        [380].S.BITS1.2   // 8-RED-760 Conf. Marcha
        [380].S.BITS1.4   // 8-RED-760 Cmd. Automatico
        [380].S.BITS1.26   // 8-RED-760 FLL
        [380].S.BITS1.27   // 8-RED-760 FV0
        [380].S.BITS1.28   // 8-RED-760 FATO
        [380].S.BITS1.30   // 8-RED-760 Falla Partida
        [380].S.BITS2.20   // 8-RED-760 Reset Falla
        [380].S.BITS2.23   // 8-RED-760 Test
        [380].S.BITS2.27   // 8-RED-760 Cmd. Marcha
        [380].S.BITS2.30   // 8-RED-760 OUT MARCHA
        [684].S.BITS1.29   // 120-CAN-070 Falla Abrir
        [385].S.BITS1.0   // 110-ENF-001/1-2 Enable
        [442].S.BITS1.9   // 9-BIN-704 LM
        [632].S.BITS1.9   // 120-CAN-022 Conf. Cerrado
        [405].S.BITS1.0   // 9-CON-667 Enable
        [445].S.BITS1.0   // 9-CON-707 Enable
        [304].S.BITS1.9   // 100-BCE-005 Sobrecarga
        [684].S.BITS2.20   // 120-CAN-070 Reset Falla
        [634].S.BITS1.9   // 120-CAN-023 Conf. Cerrado
        [444].S.BITS1.9   // 9-BIN-706 LM
        [382].S.BITS1.29   // 90-CAN-002 Falla Abrir
        [25].S.BITS1.2   // 7-CON-1025 Conf Pos Abrir
        [465].S.BITS1.0   // 9-CON-727 Enable
        [552].S.BITS1.8   // 110-TDC-004/1 Atollo
        [554].S.BITS1.8   // 110-ELV-001/1 Atollo
        [382].S.BITS2.31   // 110-ENF-001/1-4 OUT MARCHA
        [42].S.BITS1.2   // 7-FLT-1066 Conf. Marcha
        [515].S.BITS1.0   // 110-ENF-001/3-2 Enable
        [449].S.BITS1.9   // 110-VAL-001/2-1 Sobrecarga
        [636].S.BITS1.9   // 120-CAN-024 Conf. Cerrado
        [535].S.BITS1.0   // 110-ENF-002/3-2 Enable
        [558].S.BITS2.31   // 120-TDC-002 OUT MARCHA
        [308].S.BITS1.9   // 100-BCE-002 Sobrecarga
        [385].S.BITS1.24   // por confirmar
        [385].S.BITS1.26   // L3-QRA-010a FLL
        [385].S.BITS1.27   // L3-QRA-010a FV0
        [385].S.BITS1.28   // L3-QRA-010a FATO
        [386].S.BITS1.0   // 9-RED-650 Enable
        [386].S.BITS1.1   // 9-RED-650 Falla Resumen
        [386].S.BITS1.2   // 9-RED-650 Conf. Marcha
        [386].S.BITS1.4   // 9-RED-650 Cmd. Automatico
        [386].S.BITS1.24   // por confirmar
        [386].S.BITS1.26   // 9-RED-650 FLL
        [386].S.BITS1.27   // 9-RED-650 FV0
        [386].S.BITS1.28   // 9-RED-650 FATO
        [386].S.BITS1.29   // 90-CAN-004 Falla Abrir
        [386].S.BITS1.30   // 9-RED-650 Falla Partida
        [386].S.BITS2.20   // 9-RED-650 Reset Falla
        [386].S.BITS2.23   // 9-RED-650 Test
        [386].S.BITS2.30   // 9-RED-650 OUT MARCHA
        [386].S.BITS2.31   // 90-CAN-004 OUT OPEN
        [52].S.BITS1.2   // 7-CON-1075 Conf Pos Abrir
        [638].S.BITS1.9   // 120-CAN-025 Conf. Cerrado
        [451].S.BITS1.9   // 110-ENF-001/2-5 Sobrecarga
        [387].S.BITS1.29   // 9-CON-651 Falla Abrir
        [61].S.BITS1.2   // 7-MRO-1083a Conf. Marcha
        [566].S.BITS2.31   // 120-HAR-002 OUT MARCHA
        [555].S.BITS1.8   // 120-TDC-001/1 Atollo
        [558].S.BITS1.8   // 120-TDC-002 Atollo
        [388].S.BITS1.0   // 9-CON-652 Enable
        [388].S.BITS1.1   // 9-CON-652 Falla Resumen
        [388].S.BITS1.4   // 9-CON-652 Conf Pos Cerrar
        [388].S.BITS1.26   // L3-ELV-016 FLL
        [388].S.BITS1.27   // L3-ELV-016 FV0
        [388].S.BITS1.28   // L3-ELV-016 FATO
        [388].S.BITS1.30   // 9-CON-652 Falla Cerrar
        [388].S.BITS2.20   // 9-CON-652 Reset Falla
        [388].S.BITS2.23   // 9-CON-652 Test
        [388].S.BITS2.27   // 9-CON-652 Cmd. Open
        [388].S.BITS2.30   // 9-CON-652 OUT CLOSE
        [71].S.BITS1.2   // 90-CAN-017 Conf Pos Abrir
        [568].S.BITS2.31   // 120-TDC-003 OUT MARCHA
        [462].S.BITS1.9   // 9-BIN-724 LM
        [389].S.BITS1.29   // 9-CON-653 Falla Abrir
        [640].S.BITS1.9   // 120-CAN-026 Conf. Cerrado
        [570].S.BITS1.2   // CV-12 Conf Pos Abrir
        [389].S.BITS2.26   // Cmd. Pos . Izquierda
        [570].S.BITS1.4   // CV-12 Conf Pos Cerrar
        [312].S.BITS1.9   // 100-BCE-001 Sobrecarga
        [389].S.BITS2.31   // 9-CON-653 OUT OPEN
        [233].S.BITS1.29   // 7-LMG-1187 Falla Abrir
        [642].S.BITS1.9   // 120-CAN-033 Conf. Cerrado
        [464].S.BITS1.9   // 9-BIN-726 LM
        [390].S.BITS1.29   // 9-CON-654 Falla Abrir
        [233].S.BITS2.20   // 7-LMG-1187 Reset Falla
        [570].S.BITS1.30   // CV-12 Falla Cerrar
        [561].S.BITS1.8   // 110-TDC-003/2 Atollo
        [562].S.BITS1.8   // 110-TDC-004/2 Atollo
        [390].S.BITS2.31   // 9-CON-654 OUT OPEN
        [234].S.BITS1.29   // 100-CAN-023 Falla Abrir
        [644].S.BITS1.9   // 120-CAN-034 Conf. Cerrado
        [469].S.BITS1.9   // 110-VAL-002/2-1 Sobrecarga
        [391].S.BITS1.29   // 90-CAN-009 Falla Abrir
        [234].S.BITS2.20   // 100-CAN-023 Reset Falla
        [576].S.BITS2.31   // 120-HAR-003 OUT MARCHA
        [564].S.BITS1.8   // 110-ELV-001/2 Atollo
        [565].S.BITS1.8   // 120-TDC-001/2 Atollo
        [392].S.BITS1.0   // 9-RED-655 Enable
        [392].S.BITS1.1   // 9-RED-655 Falla Resumen
        [392].S.BITS1.2   // 9-RED-655 Conf. Marcha
        [392].S.BITS1.4   // 9-RED-655 Cmd. Automatico
        [392].S.BITS1.29   // 90-CAN-010 Falla Abrir
        [392].S.BITS1.30   // 9-RED-655 Falla Partida
        [392].S.BITS2.20   // 9-RED-655 Reset Falla
        [392].S.BITS2.23   // 9-RED-655 Test
        [392].S.BITS2.30   // 9-RED-655 OUT MARCHA
        [392].S.BITS2.31   // 90-CAN-010 OUT OPEN
        [394].S.BITS1.0   // 9-CON-657 Enable
        [394].S.BITS1.1   // 9-CON-657 Falla Resumen
        [394].S.BITS1.4   // 9-CON-657 Conf Pos Cerrar
        [394].S.BITS1.8   // TOL-VIR-010 LL
        [394].S.BITS1.9   // TOL-VIR-010 LM
        [394].S.BITS1.10   // TOL-VIR-010 LH
        [394].S.BITS1.26   // 90-TDC-005 FLL
        [394].S.BITS1.27   // 90-TDC-005 FV0
        [394].S.BITS1.28   // 90-TDC-005 FATO
        [394].S.BITS1.30   // 9-CON-657 Falla Cerrar
        [394].S.BITS2.20   // 9-CON-657 Reset Falla
        [394].S.BITS2.23   // 9-CON-657 Test
        [394].S.BITS2.27   // 9-CON-657 Cmd. Open
        [394].S.BITS2.30   // 9-CON-657 OUT CLOSE
        [395].S.BITS1.0   // 9-CON-658 Enable
        [395].S.BITS1.1   // 9-CON-658 Falla Resumen
        [395].S.BITS1.2   // 9-CON-658 Conf Pos Abrir
        [395].S.BITS1.4   // 9-CON-658 Conf Pos Cerrar
        [395].S.BITS1.29   // 9-CON-658 Falla Abrir
        [395].S.BITS1.30   // 9-CON-658 Falla Cerrar
        [395].S.BITS2.20   // 9-CON-658 Reset Falla
        [395].S.BITS2.23   // 9-CON-658 Test
        [395].S.BITS2.27   // 9-CON-658 Cmd. Open
        [395].S.BITS2.30   // 9-CON-658 OUT CLOSE
        [395].S.BITS2.31   // 9-CON-658 OUT OPEN
        [397].S.BITS1.0   // 90-TDC-006 Enable
        [397].S.BITS1.1   // 90-TDC-006 Falla Resumen
        [397].S.BITS1.2   // 90-TDC-006 Conf. Marcha
        [397].S.BITS1.4   // 90-TDC-006 Cmd. Automatico
        [397].S.BITS1.26   // 90-TDC-006 FLL
        [397].S.BITS1.27   // 90-TDC-006 FV0
        [397].S.BITS1.28   // 90-TDC-006 FATO
        [397].S.BITS1.30   // 90-TDC-006 Falla Partida
        [397].S.BITS2.20   // 90-TDC-006 Reset Falla
        [397].S.BITS2.23   // 90-TDC-006 Test
        [397].S.BITS2.27   // 90-TDC-006 Cmd. Marcha
        [397].S.BITS2.30   // 90-TDC-006 OUT MARCHA
        [398].S.BITS1.0   // 9-RED-660 Enable
        [398].S.BITS1.1   // 9-RED-660 Falla Resumen
        [398].S.BITS1.2   // 9-RED-660 Conf. Marcha
        [398].S.BITS1.4   // 9-RED-660 Cmd. Automatico
        [398].S.BITS1.29   // 90-CAN-012 Falla Abrir
        [398].S.BITS1.30   // 9-RED-660 Falla Partida
        [398].S.BITS2.20   // 9-RED-660 Reset Falla
        [398].S.BITS2.23   // 9-RED-660 Test
        [398].S.BITS2.30   // 9-RED-660 OUT MARCHA
        [398].S.BITS2.31   // 90-CAN-012 OUT OPEN
        [399].S.BITS1.0   // 9-CON-661 Enable
        [399].S.BITS1.1   // 9-CON-661 Falla Resumen
        [399].S.BITS1.2   // 9-CON-661 Conf Pos Abrir
        [399].S.BITS1.4   // 9-CON-661 Conf Pos Cerrar
        [399].S.BITS1.29   // 9-CON-661 Falla Abrir
        [399].S.BITS1.30   // 9-CON-661 Falla Cerrar
        [399].S.BITS2.20   // 9-CON-661 Reset Falla
        [399].S.BITS2.23   // 9-CON-661 Test
        [399].S.BITS2.26   // L4-BIF-044 Cmd. Pos . Izquierda
        [399].S.BITS2.27   // 9-CON-661 Cmd. Open
        [399].S.BITS2.30   // 9-CON-661 OUT CLOSE
        [399].S.BITS2.31   // 9-CON-661 OUT OPEN
        [400].S.BITS1.0   // 9-CON-662 Enable
        [400].S.BITS1.1   // 9-CON-662 Falla Resumen
        [400].S.BITS1.4   // 9-CON-662 Conf Pos Cerrar
        [400].S.BITS1.26   // 90-TDC-007 FLL
        [400].S.BITS1.27   // 90-TDC-007 FV0
        [400].S.BITS1.28   // 90-TDC-007 FATO
        [400].S.BITS1.30   // 9-CON-662 Falla Cerrar
        [400].S.BITS2.20   // 9-CON-662 Reset Falla
        [400].S.BITS2.23   // 9-CON-662 Test
        [400].S.BITS2.27   // 9-CON-662 Cmd. Open
        [400].S.BITS2.30   // 9-CON-662 OUT CLOSE
        [235].S.BITS1.29   // 100-CAN-024 Falla Abrir
        [646].S.BITS1.9   // 120-CAN-035 Conf. Cerrado
        [471].S.BITS1.9   // 110-ENF-002/2-5 Sobrecarga
        [401].S.BITS1.29   // 9-CON-663 Falla Abrir
        [235].S.BITS2.20   // 7-LRT-1189 Reset Falla
        [581].S.BITS2.31   // 120-TDC-005 OUT MARCHA
        [566].S.BITS1.8   // 120-HAR-002 Atollo
        [568].S.BITS1.8   // 120-TDC-003 Atollo
        [401].S.BITS2.31   // 9-CON-663 OUT OPEN
        [236].S.BITS1.29   // 100-CAN-025 Falla Abrir
        [648].S.BITS1.9   // 120-CAN-036 Conf. Cerrado
        [512].S.BITS1.9   // 110-ENF-001/3-4 Sobrecarga
        [402].S.BITS1.29   // 9-CON-664 Falla Abrir
        [236].S.BITS2.20   // 100-CAN-025 Reset Falla
        [591].S.BITS2.31   // 120-TDC-006 OUT MARCHA
        [571].S.BITS1.8   // 110-TDC-003/3 Atollo
        [572].S.BITS1.8   // 110-TDC-004/3 Atollo
        [403].S.BITS1.0   // 9-CON-665 Enable
        [403].S.BITS1.1   // 9-CON-665 Falla Resumen
        [403].S.BITS1.2   // 9-CON-665 Conf Pos Abrir
        [403].S.BITS1.4   // 9-CON-665 Conf Pos Cerrar
        [403].S.BITS1.26   // L4-ELV-035 FLL
        [403].S.BITS1.27   // L4-ELV-035 FV0
        [403].S.BITS1.28   // L4-ELV-035 FATO
        [403].S.BITS1.29   // 9-CON-665 Falla Abrir
        [403].S.BITS1.30   // 9-CON-665 Falla Cerrar
        [403].S.BITS2.20   // 9-CON-665 Reset Falla
        [403].S.BITS2.23   // 9-CON-665 Test
        [403].S.BITS2.27   // 9-CON-665 Cmd. Open
        [403].S.BITS2.30   // 9-CON-665 OUT CLOSE
        [403].S.BITS2.31   // 9-CON-665 OUT OPEN
        [297].S.BITS2.27   // 100-TOL-003-1 Cmd. Open
        [650].S.BITS1.9   // 120-CAN-037 Conf. Cerrado
        [514].S.BITS1.9   // 110-ENF-001/3-1 Sobrecarga
        [404].S.BITS1.29   // 9-CON-666 Falla Abrir
        [297].S.BITS2.30   // 100-TOL-003-1 OUT CLOSE
        [601].S.BITS2.31   // 120-TDC-007 OUT MARCHA
        [573].S.BITS1.8   // 110-TDC-005/3 Atollo
        [574].S.BITS1.8   // 110-ELV-001/3 Atollo
        [406].S.BITS1.0   // 9-CON-668 Enable
        [406].S.BITS1.1   // 9-CON-668 Falla Resumen
        [406].S.BITS1.4   // 9-CON-668 Conf Pos Cerrar
        [406].S.BITS1.26   // L4-ZDA-037 FLL
        [406].S.BITS1.27   // L4-ZDA-037 FV0
        [406].S.BITS1.28   // L4-ZDA-037 FATO
        [406].S.BITS1.30   // 9-CON-668 Falla Cerrar
        [406].S.BITS2.20   // 9-CON-668 Reset Falla
        [406].S.BITS2.23   // 9-CON-668 Test
        [406].S.BITS2.27   // 9-CON-668 Cmd. Open
        [406].S.BITS2.30   // 9-CON-668 OUT CLOSE
        [299].S.BITS2.31   // 100-TDP-006 OUT MARCHA
        [611].S.BITS2.31   // 120-TDC-008 OUT MARCHA
        [519].S.BITS1.9   // 110-VAL-001/3-1 Sobrecarga
        [407].S.BITS1.29   // L4-BIF-045 Falla Pos. Izquierda
        [652].S.BITS1.9   // 120-CAN-038 Conf. Cerrado
        [678].S.BITS2.30   // 120-CAN-067 OUT CLOSE
        [407].S.BITS2.26   // L4-BIF-045 Cmd. Pos . Izquierda
        [678].S.BITS2.31   // 120-CAN-067 OUT OPEN
        [314].S.BITS1.8   // 100-VEN-ACORG-1 Atollo
        [408].S.BITS1.0   // 9-RED-670 Enable
        [408].S.BITS1.1   // 9-RED-670 Falla Resumen
        [408].S.BITS1.2   // 9-RED-670 Conf. Marcha
        [408].S.BITS1.4   // 9-RED-670 Cmd. Automatico
        [408].S.BITS1.29   // 90-CAN-022 Falla Abrir
        [408].S.BITS1.30   // 9-RED-670 Falla Partida
        [408].S.BITS2.20   // 9-RED-670 Reset Falla
        [408].S.BITS2.23   // 9-RED-670 Test
        [408].S.BITS2.30   // 9-RED-670 OUT MARCHA
        [408].S.BITS2.31   // 90-CAN-022 OUT OPEN
        [654].S.BITS1.9   // 120-CAN-047 Conf. Cerrado
        [521].S.BITS1.9   // 110-ENF-001/3-5 Sobrecarga
        [409].S.BITS1.29   // 9-CON-671 Falla Abrir
        [680].S.BITS2.30   // 120-CAN-068 OUT CLOSE
        [575].S.BITS1.8   // 120-TDC-001/3 Atollo
        [576].S.BITS1.8   // 120-HAR-003 Atollo
        [409].S.BITS2.31   // 9-CON-671 OUT OPEN
        [656].S.BITS1.9   // 120-CAN-048 Conf. Cerrado
        [532].S.BITS1.9   // 110-ENF-002/3-4 Sobrecarga
        [410].S.BITS1.29   // 9-CON-672 Falla Abrir
        [680].S.BITS2.31   // 120-CAN-068 OUT OPEN
        [581].S.BITS1.8   // 120-TDC-005 Atollo
        [591].S.BITS1.8   // 120-TDC-006 Atollo
        [410].S.BITS2.31   // 9-CON-672 OUT OPEN
        [658].S.BITS1.9   // 120-CAN-049 Conf. Cerrado
        [534].S.BITS1.9   // 110-ENF-002/3-1 Sobrecarga
        [411].S.BITS1.29   // 9-CON-673 Falla Abrir
        [682].S.BITS2.30   // 120-CAN-069 OUT CLOSE
        [601].S.BITS1.8   // 120-TDC-007 Atollo
        [611].S.BITS1.8   // 120-TDC-008 Atollo
        [412].S.BITS1.0   // 9-CON-674 Enable
        [412].S.BITS1.1   // 9-CON-674 Falla Resumen
        [412].S.BITS1.2   // 9-CON-674 Conf Pos Abrir
        [412].S.BITS1.4   // 9-CON-674 Conf Pos Cerrar
        [412].S.BITS1.26   // 75-TDC-003 FLL
        [412].S.BITS1.27   // 75-TDC-003 FV0
        [412].S.BITS1.28   // 75-TDC-003 FATO
        [412].S.BITS1.29   // 9-CON-674 Falla Abrir
        [412].S.BITS1.30   // 9-CON-674 Falla Cerrar
        [412].S.BITS2.20   // 9-CON-674 Reset Falla
        [412].S.BITS2.23   // 9-CON-674 Test
        [412].S.BITS2.27   // 9-CON-674 Cmd. Open
        [412].S.BITS2.30   // 9-CON-674 OUT CLOSE
        [412].S.BITS2.31   // 9-CON-674 OUT OPEN
        [413].S.BITS1.0   // 9-CON-675 Enable
        [413].S.BITS1.1   // 9-CON-675 Falla Resumen
        [413].S.BITS1.2   // 9-CON-675 Conf Pos Abrir
        [413].S.BITS1.4   // 9-CON-675 Conf Pos Cerrar
        [413].S.BITS1.29   // 9-CON-675 Falla Abrir
        [413].S.BITS1.30   // 9-CON-675 Falla Cerrar
        [413].S.BITS2.20   // 9-CON-675 Reset Falla
        [413].S.BITS2.23   // 9-CON-675 Test
        [413].S.BITS2.27   // 9-CON-675 Cmd. Open
        [413].S.BITS2.30   // 9-CON-675 OUT CLOSE
        [413].S.BITS2.31   // 9-CON-675 OUT OPEN
        [682].S.BITS2.31   // 120-CAN-069 OUT OPEN
        [539].S.BITS1.9   // 110-VEN-002/3-1 Sobrecarga
        [660].S.BITS1.9   // 120-CAN-050 Conf. Cerrado
        [684].S.BITS2.30   // 120-CAN-070 OUT CLOSE
        [684].S.BITS2.31   // 120-CAN-070 OUT OPEN
        [315].S.BITS1.8   // 100-VEN-ACORG-2 Atollo
        [662].S.BITS1.9   // 120-CAN-051 Conf. Cerrado
        [541].S.BITS1.9   // 110-ENF-002/3-5 Sobrecarga
        [415].S.BITS1.29   // 9-CON-677 Falla Abrir
        [678].S.BITS1.0   // 120-CAN-067 Enable
        [680].S.BITS1.0   // 120-CAN-068 Enable
        [415].S.BITS2.31   // 9-CON-677 OUT OPEN
        [664].S.BITS1.9   // 120-CAN-052 Conf. Cerrado
        [557].S.BITS1.10   // 120-XY-8127 Conf. Abierto
        [416].S.BITS1.29   // 9-CON-678 Falla Abrir
        [682].S.BITS1.0   // 120-CAN-069 Enable
        [684].S.BITS1.0   // 120-CAN-070 Enable
        [416].S.BITS2.31   // 9-CON-678 OUT OPEN
        [666].S.BITS1.9   // 120-CAN-053 Conf. Cerrado
        [559].S.BITS1.10   // 120-CAN-001 Conf. Abierto
        [417].S.BITS1.29   // 90-CAN-023 Falla Abrir
        [25].S.BITS2.27   // 7-CON-1025 Cmd. Open
        [417].S.BITS2.31   // 110-TOL-006/1 OUT MARCHA
        [668].S.BITS1.9   // 120-CAN-054 Conf. Cerrado
        [567].S.BITS1.10   // 120-XY-8128 Conf. Abierto
        [418].S.BITS1.29   // 90-CAN-024 Falla Abrir
        [25].S.BITS2.30   // 7-CON-1025 OUT CLOSE
        [26].S.BITS2.31   // 7-CON-1026 OUT OPEN
        [419].S.BITS1.0   // 9-CON-681 Enable
        [419].S.BITS1.1   // 9-CON-681 Falla Resumen
        [419].S.BITS1.2   // 9-CON-681 Conf Pos Abrir
        [419].S.BITS1.4   // 9-CON-681 Conf Pos Cerrar
        [419].S.BITS1.26   // 90-TDC-017 FLL
        [419].S.BITS1.27   // 90-TDC-017 FV0
        [419].S.BITS1.28   // 90-TDC-017 FATO
        [419].S.BITS1.29   // 9-CON-681 Falla Abrir
        [419].S.BITS1.30   // 9-CON-681 Falla Cerrar
        [419].S.BITS2.20   // 9-CON-681 Reset Falla
        [419].S.BITS2.23   // 9-CON-681 Test
        [419].S.BITS2.27   // 9-CON-681 Cmd. Open
        [419].S.BITS2.30   // 9-CON-681 OUT CLOSE
        [419].S.BITS2.31   // 9-CON-681 OUT OPEN
        [420].S.BITS1.0   // 9-CON-682 Enable
        [420].S.BITS1.1   // 9-CON-682 Falla Resumen
        [420].S.BITS1.2   // 9-CON-682 Conf Pos Abrir
        [420].S.BITS1.4   // 9-CON-682 Conf Pos Cerrar
        [420].S.BITS1.29   // 9-CON-682 Falla Abrir
        [420].S.BITS1.30   // 9-CON-682 Falla Cerrar
        [420].S.BITS2.20   // 9-CON-682 Reset Falla
        [420].S.BITS2.23   // 9-CON-682 Test
        [420].S.BITS2.27   // 9-CON-682 Cmd. Open
        [420].S.BITS2.30   // 9-CON-682 OUT CLOSE
        [420].S.BITS2.31   // 9-CON-682 OUT OPEN
        [421].S.BITS1.0   // 9-CON-683 Enable
        [421].S.BITS1.1   // 9-CON-683 Falla Resumen
        [421].S.BITS1.4   // 9-CON-683 Conf Pos Cerrar
        [421].S.BITS1.26   // 90-TDC-010 FLL
        [421].S.BITS1.27   // 90-TDC-010 FV0
        [421].S.BITS1.28   // 90-TDC-010 FATO
        [421].S.BITS1.29   // 9-CON-683 Falla Abrir
        [421].S.BITS1.30   // 9-CON-683 Falla Cerrar
        [421].S.BITS2.20   // 9-CON-683 Reset Falla
        [421].S.BITS2.23   // 9-CON-683 Test
        [421].S.BITS2.27   // 9-CON-683 Cmd. Open
        [421].S.BITS2.30   // 9-CON-683 OUT CLOSE
        [421].S.BITS2.31   // 9-CON-683 OUT OPEN
        [422].S.BITS1.0   // 9-CON-684 Enable
        [422].S.BITS1.1   // 9-CON-684 Falla Resumen
        [422].S.BITS1.2   // 9-CON-684 Conf Pos Abrir
        [422].S.BITS1.4   // 9-CON-684 Conf Pos Cerrar
        [422].S.BITS1.29   // 9-CON-684 Falla Abrir
        [422].S.BITS1.30   // 9-CON-684 Falla Cerrar
        [422].S.BITS2.20   // 9-CON-684 Reset Falla
        [422].S.BITS2.23   // 9-CON-684 Test
        [422].S.BITS2.27   // 9-CON-684 Cmd. Open
        [422].S.BITS2.30   // 9-CON-684 OUT CLOSE
        [422].S.BITS2.31   // 9-CON-684 OUT OPEN
        [670].S.BITS1.9   // 120-CAN-063 Conf. Cerrado
        [569].S.BITS1.10   // 120-CAN-003 Conf. Abierto
        [28].S.BITS2.31   // 90-VEN-006 OUT MARCHA
        [29].S.BITS2.31   // 90-TDC-005 OUT MARCHA
        [461].S.BITS1.8   // 110-ESC-002/2 Atollo
        [672].S.BITS1.9   // 120-CAN-064 Conf. Cerrado
        [577].S.BITS1.10   // 120-XY-8129 Conf. Abierto
        [40].S.BITS2.31   // 90-TAB-001 OUT MARCHA
        [467].S.BITS1.8   // 110-ESC-004/2 Atollo
        [674].S.BITS1.9   // 120-CAN-065 Conf. Cerrado
        [582].S.BITS1.10   // 120-CAN-007 Conf. Abierto
        [425].S.BITS1.29   // 9-CON-687 Falla Abrir
        [42].S.BITS2.31   // 90-CAN-013 OUT OPEN
        [43].S.BITS2.31   // 90-ALI-001 OUT MARCHA
        [426].S.BITS1.0   // 9-CON-688 Enable
        [426].S.BITS1.1   // 9-CON-688 Falla Resumen
        [426].S.BITS1.2   // 9-CON-688 Conf Pos Abrir
        [426].S.BITS1.4   // 9-CON-688 Conf Pos Cerrar
        [426].S.BITS1.29   // 9-CON-688 Falla Abrir
        [426].S.BITS1.30   // 9-CON-688 Falla Cerrar
        [426].S.BITS2.20   // 9-CON-688 Reset Falla
        [426].S.BITS2.23   // 9-CON-688 Test
        [426].S.BITS2.27   // 9-CON-688 Cmd. Open
        [426].S.BITS2.30   // 9-CON-688 OUT CLOSE
        [426].S.BITS2.31   // 9-CON-688 OUT OPEN
        [427].S.BITS1.0   // 90-TDC-018 Enable
        [427].S.BITS1.1   // 90-TDC-018 Falla Resumen
        [427].S.BITS1.2   // 90-TDC-018 Conf. Marcha
        [427].S.BITS1.4   // 90-TDC-018 Cmd. Automatico
        [427].S.BITS1.26   // 90-TDC-018 FLL
        [427].S.BITS1.27   // 90-TDC-018 FV0
        [427].S.BITS1.28   // 90-TDC-018 FATO
        [427].S.BITS1.30   // 90-TDC-018 Falla Partida
        [427].S.BITS2.20   // 90-TDC-018 Reset Falla
        [427].S.BITS2.23   // 90-TDC-018 Test
        [427].S.BITS2.27   // 90-TDC-018 Cmd. Marcha
        [427].S.BITS2.30   // 90-TDC-018 OUT MARCHA
        [428].S.BITS1.0   // 9-RED-690 Enable
        [428].S.BITS1.1   // 9-RED-690 Falla Resumen
        [428].S.BITS1.2   // 9-RED-690 Conf. Marcha
        [428].S.BITS1.4   // 9-RED-690 Cmd. Automatico
        [428].S.BITS1.26   // 9-RED-690 FLL
        [428].S.BITS1.27   // 9-RED-690 FV0
        [428].S.BITS1.28   // 9-RED-690 FATO
        [428].S.BITS1.29   // 90-CAN-093 Falla Abrir
        [428].S.BITS1.30   // 9-RED-690 Falla Partida
        [428].S.BITS2.20   // 9-RED-690 Reset Falla
        [428].S.BITS2.23   // 9-RED-690 Test
        [428].S.BITS2.27   // 9-RED-690 Cmd. Marcha
        [428].S.BITS2.30   // 9-RED-690 OUT MARCHA
        [428].S.BITS2.31   // 90-CAN-093 OUT OPEN
        [429].S.BITS1.0   // 9-CON-691 Enable
        [429].S.BITS1.1   // 9-CON-691 Falla Resumen
        [429].S.BITS1.2   // 9-CON-691 Conf Pos Abrir
        [429].S.BITS1.4   // 9-CON-691 Conf Pos Cerrar
        [429].S.BITS1.29   // 9-CON-691 Falla Abrir
        [429].S.BITS1.30   // 9-CON-691 Falla Cerrar
        [429].S.BITS2.20   // 9-CON-691 Reset Falla
        [429].S.BITS2.23   // 9-CON-691 Test
        [429].S.BITS2.27   // 9-CON-691 Cmd. Open
        [429].S.BITS2.30   // 9-CON-691 OUT CLOSE
        [429].S.BITS2.31   // 9-CON-691 OUT OPEN
        [676].S.BITS1.9   // 120-CAN-066 Conf. Cerrado
        [583].S.BITS1.10   // 120-CAN-008 Conf. Abierto
        [430].S.BITS1.29   // 9-CON-692 Falla Abrir
        [46].S.BITS2.31   // 90-MMA-001 OUT MARCHA
        [49].S.BITS2.31   // 7-CON-1072 OUT OPEN
        [431].S.BITS1.0   // 9-CON-693 Enable
        [431].S.BITS1.1   // 9-CON-693 Falla Resumen
        [431].S.BITS1.2   // 9-CON-693 Conf Pos Abrir
        [431].S.BITS1.4   // 9-CON-693 Conf Pos Cerrar
        [431].S.BITS1.29   // 9-CON-693 Falla Abrir
        [431].S.BITS1.30   // 9-CON-693 Falla Cerrar
        [431].S.BITS2.20   // 9-CON-693 Reset Falla
        [431].S.BITS2.23   // 9-CON-693 Test
        [431].S.BITS2.27   // 9-CON-693 Cmd. Open
        [431].S.BITS2.30   // 9-CON-693 OUT CLOSE
        [431].S.BITS2.31   // 9-CON-693 OUT OPEN
        [678].S.BITS1.1   // 120-CAN-067 Falla Resumen
        [584].S.BITS1.10   // 120-CAN-009 Conf. Abierto
        [432].S.BITS1.29   // 9-CON-694 Falla Abrir
        [50].S.BITS2.31   // 7-CON-1073 OUT OPEN
        [52].S.BITS2.30   // 7-CON-1075 OUT CLOSE
        [432].S.BITS2.31   // 9-CON-694 OUT OPEN
        [585].S.BITS1.10   // 120-CAN-010 Conf. Abierto
        [678].S.BITS1.9   // 120-CAN-067 Conf. Cerrado
        [323].S.BITS1.9   // 100-VIB-001 Sobrecarga
        [678].S.BITS1.30   // 120-CAN-067 Falla Cerrar
        [586].S.BITS1.10   // 120-CAN-011 Conf. Abierto
        [434].S.BITS1.29   // 9-CON-696 Falla Abrir
        [52].S.BITS2.31   // 7-CON-1075 OUT OPEN
        [53].S.BITS2.31   // 90-CAN-015 OUT OPEN
        [434].S.BITS2.31   // 9-CON-696 OUT OPEN
        [680].S.BITS1.1   // 120-CAN-068 Falla Resumen
        [587].S.BITS1.10   // 120-CAN-012 Conf. Abierto
        [435].S.BITS1.29   // 9-CON-697 Falla Abrir
        [54].S.BITS2.31   // 7-CON-1077 OUT OPEN
        [56].S.BITS2.31   // 7-CON-1079 OUT OPEN
        [435].S.BITS2.31   // 9-CON-697 OUT OPEN
        [680].S.BITS1.9   // 120-CAN-068 Conf. Cerrado
        [588].S.BITS1.10   // 120-CAN-013 Conf. Abierto
        [436].S.BITS1.29   // 9-CON-698 Falla Abrir
        [57].S.BITS2.31   // 7-CON-1080 OUT OPEN
        [59].S.BITS2.31   // 90-TOR-002 OUT MARCHA
        [437].S.BITS1.8   // 90-SIL-010 LL
        [438].S.BITS1.0   // 90-TDC-013 Enable
        [438].S.BITS1.1   // 90-TDC-013 Falla Resumen
        [438].S.BITS1.2   // 90-TDC-013 Conf. Marcha
        [438].S.BITS1.4   // 90-TDC-013 Cmd. Automatico
        [438].S.BITS1.8   // 9-BIN-700 LL
        [438].S.BITS1.9   // 9-BIN-700 LM
        [438].S.BITS1.10   // 9-BIN-700 LH
        [438].S.BITS1.26   // 90-TDC-013 FLL
        [438].S.BITS1.27   // 90-TDC-013 FV0
        [438].S.BITS1.28   // 90-TDC-013 FATO
        [438].S.BITS1.30   // 90-TDC-013 Falla Partida
        [438].S.BITS2.20   // 90-TDC-013 Reset Falla
        [438].S.BITS2.23   // 90-TDC-013 Test
        [438].S.BITS2.27   // 90-TDC-013 Cmd. Marcha
        [438].S.BITS2.30   // 90-TDC-013 OUT MARCHA
        [439].S.BITS1.0   // 9-CON-701 Enable
        [439].S.BITS1.1   // 9-CON-701 Falla Resumen
        [439].S.BITS1.2   // 9-CON-701 Conf Pos Abrir
        [439].S.BITS1.4   // 9-CON-701 Conf Pos Cerrar
        [439].S.BITS1.8   // 90-SIL-008 LL
        [439].S.BITS1.9   // 90-SIL-008 LM
        [439].S.BITS1.10   // 90-SIL-008 LH
        [439].S.BITS1.29   // 9-CON-701 Falla Abrir
        [439].S.BITS1.30   // 9-CON-701 Falla Cerrar
        [439].S.BITS2.20   // 9-CON-701 Reset Falla
        [439].S.BITS2.23   // 9-CON-701 Test
        [439].S.BITS2.27   // 9-CON-701 Cmd. Open
        [439].S.BITS2.30   // 9-CON-701 OUT CLOSE
        [439].S.BITS2.31   // 9-CON-701 OUT OPEN
        [440].S.BITS1.0   // 90-CAN-040 Enable
        [440].S.BITS1.1   // 90-CAN-040 Falla Resumen
        [440].S.BITS1.2   // 90-CAN-040 Conf Pos Abrir
        [440].S.BITS1.4   // 90-CAN-040 Conf Pos Cerrar
        [440].S.BITS1.8   // 9-BIN-702 LL
        [440].S.BITS1.9   // 9-BIN-702 LM
        [440].S.BITS1.10   // 9-BIN-702 LH
        [440].S.BITS1.29   // 90-CAN-040 Falla Abrir
        [440].S.BITS1.30   // 90-CAN-040 Falla Cerrar
        [440].S.BITS2.20   // 90-CAN-040 Reset Falla
        [440].S.BITS2.23   // 90-CAN-040 Test
        [440].S.BITS2.27   // 90-CAN-040 Cmd. Open
        [440].S.BITS2.30   // 90-CAN-040 OUT CLOSE
        [440].S.BITS2.31   // 90-CAN-040 OUT OPEN
        [680].S.BITS1.30   // 120-CAN-068 Falla Cerrar
        [589].S.BITS1.10   // 120-CAN-014 Conf. Abierto
        [441].S.BITS1.29   // 9-CON-703 Falla Abrir
        [60].S.BITS1.4   // CV-4 Conf Pos Cerrar
        [61].S.BITS2.31   // 90-CAN-016 OUT OPEN
        [441].S.BITS2.31   // 9-CON-703 OUT OPEN
        [443].S.BITS1.0   // 9-CON-705 Enable
        [443].S.BITS1.1   // 9-CON-705 Falla Resumen
        [443].S.BITS1.4   // 9-CON-705 Conf Pos Cerrar
        [443].S.BITS1.26   // 90-TDC-014 FLL
        [443].S.BITS1.27   // 90-TDC-014 FV0
        [443].S.BITS1.28   // 90-TDC-014 FATO
        [443].S.BITS1.29   // 9-CON-705 Falla Abrir
        [443].S.BITS1.30   // 9-CON-705 Falla Cerrar
        [443].S.BITS2.20   // 9-CON-705 Reset Falla
        [443].S.BITS2.23   // 9-CON-705 Test
        [443].S.BITS2.27   // 9-CON-705 Cmd. Open
        [443].S.BITS2.30   // 9-CON-705 OUT CLOSE
        [443].S.BITS2.31   // 9-CON-705 OUT OPEN
        [682].S.BITS1.1   // 120-CAN-069 Falla Resumen
        [590].S.BITS1.10   // 120-CAN-015 Conf. Abierto
        [444].S.BITS1.29   // 90-CAN-121 Falla Abrir
        [62].S.BITS2.31   // 90-ALI-003 OUT MARCHA
        [71].S.BITS2.31   // 90-CAN-017 OUT OPEN
        [446].S.BITS1.0   // 90-CAN-043 Enable
        [446].S.BITS1.1   // 90-CAN-043 Falla Resumen
        [446].S.BITS1.2   // 90-CAN-043 Conf Pos Abrir
        [446].S.BITS1.3   // 90-TRI-001 Conf. Pos. Centro
        [446].S.BITS1.4   // 90-CAN-043 Conf Pos Cerrar
        [446].S.BITS1.29   // 90-CAN-043 Falla Abrir
        [446].S.BITS1.30   // 90-CAN-043 Falla Cerrar
        [446].S.BITS2.20   // 90-CAN-043 Reset Falla
        [446].S.BITS2.23   // 90-CAN-043 Test
        [446].S.BITS2.25   // 90-TRI-001 Cmd. Pos . Izquierda
        [446].S.BITS2.26   // 90-TRI-001 Cmd. Pos . Centro
        [446].S.BITS2.27   // 90-CAN-043 Cmd. Open
        [446].S.BITS2.30   // 90-CAN-043 OUT CLOSE
        [446].S.BITS2.31   // 90-CAN-043 OUT OPEN
        [447].S.BITS1.2   // 9-CON-709 Conf Pos Abrir
        [447].S.BITS1.3   // 90-TRI-002 Conf. Pos. Centro
        [447].S.BITS1.4   // 9-CON-709 Conf Pos Cerrar
        [447].S.BITS1.29   // 9-CON-709 Falla Abrir
        [447].S.BITS1.30   // 9-CON-709 Falla Cerrar
        [447].S.BITS2.25   // 90-TRI-002 Cmd. Pos . Izquierda
        [447].S.BITS2.26   // 90-TRI-002 Cmd. Pos . Centro
        [447].S.BITS2.27   // 9-CON-709 Cmd. Open
        [324].S.BITS1.10   // XY-6103 Conf. Abierto
        [448].S.BITS1.0   // 90-BIF-LM-1 Enable
        [448].S.BITS1.1   // 90-BIF-LM-1 Falla Resumen
        [448].S.BITS1.2   // 90-BIF-LM-1 Conf. Pos. Izquierda
        [448].S.BITS1.4   // 90-BIF-LM-1 Conf. Pos. Derecha
        [448].S.BITS1.29   // 90-BIF-LM-1 Falla Pos. Izquierda
        [448].S.BITS1.30   // 90-BIF-LM-1 Falla Pos. Derecha
        [448].S.BITS2.20   // 90-BIF-LM-1 Reset Falla
        [448].S.BITS2.23   // 90-BIF-LM-1 Test
        [448].S.BITS2.26   // 90-BIF-LM-1 Cmd. Pos . Izquierda
        [448].S.BITS2.27   // 90-BIF-LM-1 Cmd. Pos. Derecha
        [448].S.BITS2.30   // 90-BIF-LM-1 Out Izquierda
        [448].S.BITS2.31   // 90-BIF-LM-1 Out Derecha
        [449].S.BITS1.2   // 9-CON-711 Conf Pos Abrir
        [196].S.BITS1.10   // 7-DOS-1170-12 LH
        [449].S.BITS1.29   // 9-CON-711 Falla Abrir
        [449].S.BITS1.30   // 9-CON-711 Falla Cerrar
        [449].S.BITS2.26   // 90-BIF-MAN Cmd. Pos . Izquierda
        [449].S.BITS2.27   // 9-CON-711 Cmd. Open
        [682].S.BITS1.9   // 120-CAN-069 Conf. Cerrado
        [449].S.BITS2.31   // 9-CON-711 OUT OPEN
        [592].S.BITS1.10   // 120-CAN-027 Conf. Abierto
        [682].S.BITS1.30   // 120-CAN-069 Falla Cerrar
        [325].S.BITS1.9   // 100-TDC-007 Sobrecarga
        [593].S.BITS1.10   // 120-CAN-028 Conf. Abierto
        [684].S.BITS1.1   // 120-CAN-070 Falla Resumen
        [326].S.BITS1.9   // 8-ENF-640 LM
        [452].S.BITS1.0   // 90-TDC-015 Enable
        [452].S.BITS1.1   // 90-TDC-015 Falla Resumen
        [452].S.BITS1.2   // 90-TDC-015 Conf. Marcha
        [452].S.BITS1.4   // 90-TDC-015 Cmd. Automatico
        [452].S.BITS1.26   // 90-TDC-015 FLL
        [452].S.BITS1.27   // 90-TDC-015 FV0
        [452].S.BITS1.28   // 90-TDC-015 FATO
        [452].S.BITS1.30   // 90-TDC-015 Falla Partida
        [452].S.BITS2.20   // 90-TDC-015 Reset Falla
        [452].S.BITS2.23   // 90-TDC-015 Test
        [452].S.BITS2.27   // 90-TDC-015 Cmd. Marcha
        [452].S.BITS2.30   // 90-TDC-015 OUT MARCHA
        [453].S.BITS1.0   // 9-CON-715 Enable
        [453].S.BITS1.1   // 9-CON-715 Falla Resumen
        [453].S.BITS1.2   // 9-CON-715 Conf Pos Abrir
        [453].S.BITS1.4   // 9-CON-715 Conf Pos Cerrar
        [453].S.BITS1.29   // 9-CON-715 Falla Abrir
        [453].S.BITS1.30   // 9-CON-715 Falla Cerrar
        [453].S.BITS2.20   // 9-CON-715 Reset Falla
        [453].S.BITS2.23   // 9-CON-715 Test
        [453].S.BITS2.27   // 9-CON-715 Cmd. Open
        [453].S.BITS2.30   // 9-CON-715 OUT CLOSE
        [453].S.BITS2.31   // 9-CON-715 OUT OPEN
        [454].S.BITS1.0   // 90-CAN-056 Enable
        [454].S.BITS1.1   // 90-CAN-056 Falla Resumen
        [454].S.BITS1.2   // 90-CAN-056 Conf Pos Abrir
        [454].S.BITS1.4   // 90-CAN-056 Conf Pos Cerrar
        [454].S.BITS1.29   // 90-CAN-056 Falla Abrir
        [454].S.BITS1.30   // 90-CAN-056 Falla Cerrar
        [454].S.BITS2.20   // 90-CAN-056 Reset Falla
        [454].S.BITS2.23   // 90-CAN-056 Test
        [454].S.BITS2.27   // 90-CAN-056 Cmd. Open
        [454].S.BITS2.30   // 90-CAN-056 OUT CLOSE
        [454].S.BITS2.31   // 90-CAN-056 OUT OPEN
        [455].S.BITS1.0   // 9-CON-717 Enable
        [455].S.BITS1.1   // 9-CON-717 Falla Resumen
        [455].S.BITS1.2   // 9-CON-717 Conf Pos Abrir
        [455].S.BITS1.4   // 9-CON-717 Conf Pos Cerrar
        [455].S.BITS1.29   // 9-CON-717 Falla Abrir
        [455].S.BITS1.30   // 9-CON-717 Falla Cerrar
        [455].S.BITS2.20   // 9-CON-717 Reset Falla
        [455].S.BITS2.23   // 9-CON-717 Test
        [455].S.BITS2.27   // 9-CON-717 Cmd. Open
        [455].S.BITS2.30   // 9-CON-717 OUT CLOSE
        [455].S.BITS2.31   // 9-CON-717 OUT OPEN
        [456].S.BITS1.0   // 90-COMV-02 Enable
        [456].S.BITS1.1   // 90-COMV-02 Falla Resumen
        [456].S.BITS1.2   // 90-COMV-02 Conf Pos Abrir
        [456].S.BITS1.4   // 90-COMV-02 Conf Pos Cerrar
        [456].S.BITS1.29   // 90-COMV-02 Falla Abrir
        [456].S.BITS1.30   // 90-COMV-02 Falla Cerrar
        [456].S.BITS2.20   // 90-COMV-02 Reset Falla
        [456].S.BITS2.23   // 90-COMV-02 Test
        [456].S.BITS2.27   // 90-COMV-02 Cmd. Open
        [456].S.BITS2.30   // 90-COMV-02 OUT CLOSE
        [456].S.BITS2.31   // 90-COMV-02 OUT OPEN
        [457].S.BITS1.0   // 9-CON-719 Enable
        [457].S.BITS1.1   // 9-CON-719 Falla Resumen
        [457].S.BITS1.2   // 9-CON-719 Conf Pos Abrir
        [457].S.BITS1.4   // 9-CON-719 Conf Pos Cerrar
        [457].S.BITS1.29   // 9-CON-719 Falla Abrir
        [457].S.BITS1.30   // 9-CON-719 Falla Cerrar
        [457].S.BITS2.20   // 9-CON-719 Reset Falla
        [457].S.BITS2.23   // 9-CON-719 Test
        [457].S.BITS2.27   // 9-CON-719 Cmd. Open
        [457].S.BITS2.30   // 9-CON-719 OUT CLOSE
        [457].S.BITS2.31   // 9-CON-719 OUT OPEN
        [458].S.BITS1.0   // 90-CAN-060 Enable
        [458].S.BITS1.1   // 90-CAN-060 Falla Resumen
        [458].S.BITS1.2   // 90-CAN-060 Conf Pos Abrir
        [458].S.BITS1.4   // 90-CAN-060 Conf Pos Cerrar
        [458].S.BITS1.29   // 90-CAN-060 Falla Abrir
        [458].S.BITS1.30   // 90-CAN-060 Falla Cerrar
        [458].S.BITS2.20   // 90-CAN-060 Reset Falla
        [458].S.BITS2.23   // 90-CAN-060 Test
        [458].S.BITS2.27   // 90-CAN-060 Cmd. Open
        [458].S.BITS2.30   // 90-CAN-060 OUT CLOSE
        [458].S.BITS2.31   // 90-CAN-060 OUT OPEN
        [459].S.BITS1.0   // 9-CON-721 Enable
        [459].S.BITS1.1   // 9-CON-721 Falla Resumen
        [459].S.BITS1.2   // 9-CON-721 Conf Pos Abrir
        [459].S.BITS1.4   // 9-CON-721 Conf Pos Cerrar
        [459].S.BITS1.29   // 9-CON-721 Falla Abrir
        [459].S.BITS1.30   // 9-CON-721 Falla Cerrar
        [459].S.BITS2.20   // 9-CON-721 Reset Falla
        [459].S.BITS2.23   // 9-CON-721 Test
        [459].S.BITS2.27   // 9-CON-721 Cmd. Open
        [459].S.BITS2.30   // 9-CON-721 OUT CLOSE
        [459].S.BITS2.31   // 9-CON-721 OUT OPEN
        [460].S.BITS1.0   // 90-TDC-017 Enable
        [460].S.BITS1.1   // 90-TDC-017 Falla Resumen
        [460].S.BITS1.2   // 90-TDC-017 Conf. Marcha
        [460].S.BITS1.4   // 90-TDC-017 Cmd. Automatico
        [460].S.BITS1.26   // 90-TDC-017 FLL
        [460].S.BITS1.27   // 90-TDC-017 FV0
        [460].S.BITS1.28   // 90-TDC-017 FATO
        [460].S.BITS1.29   // 90-CAN-062 Falla Abrir
        [460].S.BITS1.30   // 90-TDC-017 Falla Partida
        [460].S.BITS2.20   // 90-TDC-017 Reset Falla
        [460].S.BITS2.23   // 90-TDC-017 Test
        [460].S.BITS2.27   // 90-TDC-017 Cmd. Marcha
        [460].S.BITS2.30   // 90-TDC-017 OUT MARCHA
        [460].S.BITS2.31   // 90-CAN-062 OUT OPEN
        [684].S.BITS1.9   // 120-CAN-070 Conf. Cerrado
        [594].S.BITS1.10   // 120-CAN-029 Conf. Abierto
        [461].S.BITS1.29   // 9-CON-723 Falla Abrir
        [72].S.BITS2.31   // 90-ALI-004 OUT MARCHA
        [81].S.BITS2.31   // 7-CON-1094 OUT OPEN
        [461].S.BITS2.31   // 9-CON-723 OUT OPEN
        [684].S.BITS1.30   // 120-CAN-070 Falla Cerrar
        [595].S.BITS1.10   // 120-CAN-030 Conf. Abierto
        [462].S.BITS1.29   // 90-CAN-094 Falla Abrir
        [82].S.BITS2.31   // 7-CON-1095 OUT OPEN
        [92].S.BITS2.31   // 90-VEN-003 OUT MARCHA
        [463].S.BITS1.0   // 9-CON-725 Enable
        [463].S.BITS1.1   // 9-CON-725 Falla Resumen
        [463].S.BITS1.2   // 9-CON-725 Conf Pos Abrir
        [463].S.BITS1.4   // 9-CON-725 Conf Pos Cerrar
        [463].S.BITS1.29   // 9-CON-725 Falla Abrir
        [463].S.BITS1.30   // 9-CON-725 Falla Cerrar
        [463].S.BITS2.20   // 9-CON-725 Reset Falla
        [463].S.BITS2.23   // 9-CON-725 Test
        [463].S.BITS2.27   // 9-CON-725 Cmd. Open
        [463].S.BITS2.30   // 9-CON-725 OUT CLOSE
        [463].S.BITS2.31   // 9-CON-725 OUT OPEN
        [25].S.BITS1.4   // 7-CON-1025 Conf Pos Cerrar
        [596].S.BITS1.10   // 120-CAN-031 Conf. Abierto
        [464].S.BITS1.29   // 90-CAN-096 Falla Abrir
        [93].S.BITS2.31   // 90-FIL-003 OUT MARCHA
        [98].S.BITS2.31   // 90-TDC-007 OUT MARCHA
        [466].S.BITS1.0   // 90-CAN-071 Enable
        [466].S.BITS1.1   // 90-CAN-071 Falla Resumen
        [466].S.BITS1.2   // 90-CAN-071 Conf Pos Abrir
        [466].S.BITS1.4   // 90-CAN-071 Conf Pos Cerrar
        [466].S.BITS1.29   // 90-CAN-071 Falla Abrir
        [466].S.BITS1.30   // 90-CAN-071 Falla Cerrar
        [466].S.BITS2.20   // 90-CAN-071 Reset Falla
        [466].S.BITS2.23   // 90-CAN-071 Test
        [466].S.BITS2.27   // 90-CAN-071 Cmd. Open
        [466].S.BITS2.30   // 90-CAN-071 OUT CLOSE
        [466].S.BITS2.31   // 90-CAN-071 OUT OPEN
        [602].S.BITS1.10   // 120-CAN-039 Conf. Abierto
        [467].S.BITS1.29   // 9-CON-729 Falla Abrir
        [233].S.BITS1.1   // 7-LMG-1187 Falla Resumen
        [332].S.BITS1.9   // 110-FIL-001 Sobrecarga
        [468].S.BITS1.0   // 90-CAN-098 Enable
        [468].S.BITS1.1   // 90-CAN-098 Falla Resumen
        [468].S.BITS1.2   // 90-CAN-098 Conf Pos Abrir
        [468].S.BITS1.4   // 90-CAN-098 Conf Pos Cerrar
        [468].S.BITS1.29   // 90-CAN-098 Falla Abrir
        [468].S.BITS1.30   // 90-CAN-098 Falla Cerrar
        [468].S.BITS2.20   // 90-CAN-098 Reset Falla
        [468].S.BITS2.23   // 90-CAN-098 Test
        [468].S.BITS2.27   // 90-CAN-098 Cmd. Open
        [468].S.BITS2.30   // 90-CAN-098 OUT CLOSE
        [468].S.BITS2.31   // 90-CAN-098 OUT OPEN
        [234].S.BITS1.1   // 100-CAN-023 Falla Resumen
        [603].S.BITS1.10   // 120-CAN-040 Conf. Abierto
        [469].S.BITS1.29   // 9-CON-731 Falla Abrir
        [233].S.BITS2.31   // 7-LMG-1187 OUT OPEN
        [234].S.BITS2.31   // 100-CAN-023 OUT OPEN
        [469].S.BITS2.31   // 9-CON-731 OUT OPEN
        [234].S.BITS1.30   // 100-CAN-023 Falla Cerrar
        [604].S.BITS1.10   // 120-CAN-041 Conf. Abierto
        [470].S.BITS1.29   // 90-CAN-100 Falla Abrir
        [235].S.BITS2.31   // 100-CAN-024 OUT OPEN
        [236].S.BITS2.31   // 100-CAN-025 OUT OPEN
        [470].S.BITS2.31   // 110-VEN-002/2 OUT MARCHA
        [235].S.BITS1.1   // 7-LRT-1189 Falla Resumen
        [605].S.BITS1.10   // 120-CAN-042 Conf. Abierto
        [471].S.BITS1.29   // 90-CAN-101 Falla Abrir
        [288].S.BITS1.0   // 100-DOS-001-C Enable
        [288].S.BITS2.23   // 100-DOS-001-C Test
        [472].S.BITS1.0   // 90-CAN-102 Enable
        [472].S.BITS1.1   // 90-CAN-102 Falla Resumen
        [472].S.BITS1.2   // 90-CAN-102 Conf Pos Abrir
        [472].S.BITS1.4   // 90-CAN-102 Conf Pos Cerrar
        [472].S.BITS1.29   // 90-CAN-102 Falla Abrir
        [472].S.BITS1.30   // 90-CAN-102 Falla Cerrar
        [472].S.BITS2.20   // 90-CAN-102 Reset Falla
        [472].S.BITS2.23   // 90-CAN-102 Test
        [472].S.BITS2.27   // 90-CAN-102 Cmd. Open
        [472].S.BITS2.30   // 90-CAN-102 OUT CLOSE
        [472].S.BITS2.31   // 90-CAN-102 OUT OPEN
        [474]   // 90-TRI-001
        [474].S.BITS1.2   // 110-TOR-002/2 Conf. Marcha
        [474].S.BITS1.3   // 90-TRI-001 Conf. Pos. Centro
        [474].S.BITS1.4   // 110-TOR-002/2 Cmd. Automatico
        [474].S.BITS1.29   // 90-TRI-001 Falla Pos. Centro
        [474].S.BITS1.30   // 110-TOR-002/2 Falla Partida
        [474].S.BITS2.25   // 90-TRI-001 Cmd. Pos . Izquierda
        [474].S.BITS2.26   // 90-TRI-001 Cmd. Pos . Centro
        [474].S.BITS2.27   // 110-TOR-002/2 Cmd. Marcha
        [470].S.BITS1.8   // 110-VEN-002/2 Atollo
        [475]   // 90-TRI-002
        [475].S.BITS1.2   // 110-TOR-003/2 Conf. Marcha
        [475].S.BITS1.3   // 90-TRI-002 Conf. Pos. Centro
        [475].S.BITS1.4   // 110-TOR-003/2 Cmd. Automatico
        [475].S.BITS1.29   // 90-TRI-002 Falla Pos. Centro
        [475].S.BITS1.30   // 110-TOR-003/2 Falla Partida
        [475].S.BITS2.25   // 90-TRI-002 Cmd. Pos . Izquierda
        [475].S.BITS2.26   // 90-TRI-002 Cmd. Pos . Centro
        [475].S.BITS2.27   // 110-TOR-003/2 Cmd. Marcha
        [334].S.BITS1.9   // 110-FIL-002 Sobrecarga
        [476]   // 90-BIF-001
        [476].S.BITS1.2   // 110-ELV-002/2 Conf. Marcha
        [476].S.BITS1.4   // 110-ELV-002/2 Cmd. Automatico
        [476].S.BITS1.29   // 90-BIF-001 Falla Pos. Izquierda
        [476].S.BITS1.30   // 110-ELV-002/2 Falla Partida
        [476].S.BITS2.26   // 90-BIF-001 Cmd. Pos . Izquierda
        [476].S.BITS2.27   // 110-ELV-002/2 Cmd. Marcha
        [476].S.BITS2.30   // 110-ELV-002/2 OUT MARCHA
        [477].S.BITS1.0   // 90-CAN-049 Enable
        [477].S.BITS1.1   // 90-CAN-049 Falla Resumen
        [477].S.BITS1.2   // 90-CAN-049 Conf Pos Abrir
        [477].S.BITS1.4   // 90-CAN-049 Conf Pos Cerrar
        [477].S.BITS1.29   // 90-CAN-049 Falla Abrir
        [477].S.BITS1.30   // 90-CAN-049 Falla Cerrar
        [477].S.BITS2.20   // 90-CAN-049 Reset Falla
        [477].S.BITS2.23   // 90-CAN-049 Test
        [477].S.BITS2.27   // 90-CAN-049 Cmd. Open
        [477].S.BITS2.30   // 90-CAN-049 OUT CLOSE
        [477].S.BITS2.31   // 90-CAN-049 OUT OPEN
        [606].S.BITS1.10   // 120-CAN-043 Conf. Abierto
        [478].S.BITS1.29   // 90-CAN-050 Falla Abrir
        [236].S.BITS1.1   // 100-CAN-025 Falla Resumen
        [336].S.BITS1.9   // 110-FIL-003 Sobrecarga
        [479].S.BITS1.0   // 90-CAN-053 Enable
        [479].S.BITS1.1   // 90-CAN-053 Falla Resumen
        [479].S.BITS1.2   // 90-CAN-053 Conf Pos Abrir
        [479].S.BITS1.4   // 90-CAN-053 Conf Pos Cerrar
        [479].S.BITS1.29   // 90-CAN-053 Falla Abrir
        [479].S.BITS1.30   // 90-CAN-053 Falla Cerrar
        [479].S.BITS2.20   // 90-CAN-053 Reset Falla
        [479].S.BITS2.23   // 90-CAN-053 Test
        [479].S.BITS2.27   // 90-CAN-053 Cmd. Open
        [479].S.BITS2.30   // 90-CAN-053 OUT CLOSE
        [479].S.BITS2.31   // 90-CAN-053 OUT OPEN
        [480].S.BITS1.0   // 90-CAN-055 Enable
        [480].S.BITS1.1   // 90-CAN-055 Falla Resumen
        [480].S.BITS1.2   // 90-CAN-055 Conf Pos Abrir
        [480].S.BITS1.4   // 90-CAN-055 Conf Pos Cerrar
        [480].S.BITS1.29   // 90-CAN-055 Falla Abrir
        [480].S.BITS1.30   // 90-CAN-055 Falla Cerrar
        [480].S.BITS2.20   // 90-CAN-055 Reset Falla
        [480].S.BITS2.23   // 90-CAN-055 Test
        [480].S.BITS2.27   // 90-CAN-055 Cmd. Open
        [480].S.BITS2.30   // 90-CAN-055 OUT CLOSE
        [480].S.BITS2.31   // 90-CAN-055 OUT OPEN
        [481].S.BITS1.0   // 90-CAN-056 Enable
        [481].S.BITS1.1   // 90-CAN-056 Falla Resumen
        [481].S.BITS1.2   // 90-CAN-056 Conf Pos Abrir
        [481].S.BITS1.4   // 90-CAN-056 Conf Pos Cerrar
        [481].S.BITS1.29   // 90-CAN-056 Falla Abrir
        [481].S.BITS1.30   // 90-CAN-056 Falla Cerrar
        [481].S.BITS2.20   // 90-CAN-056 Reset Falla
        [481].S.BITS2.23   // 90-CAN-056 Test
        [481].S.BITS2.27   // 90-CAN-056 Cmd. Open
        [481].S.BITS2.30   // 90-CAN-056 OUT CLOSE
        [481].S.BITS2.31   // 90-CAN-056 OUT OPEN
        [482].S.BITS1.0   // 90-CAN-057 Enable
        [482].S.BITS1.1   // 90-CAN-057 Falla Resumen
        [482].S.BITS1.2   // 90-CAN-057 Conf Pos Abrir
        [482].S.BITS1.4   // 90-CAN-057 Conf Pos Cerrar
        [482].S.BITS1.29   // 90-CAN-057 Falla Abrir
        [482].S.BITS1.30   // 90-CAN-057 Falla Cerrar
        [482].S.BITS2.20   // 90-CAN-057 Reset Falla
        [482].S.BITS2.23   // 90-CAN-057 Test
        [482].S.BITS2.27   // 90-CAN-057 Cmd. Open
        [482].S.BITS2.30   // 90-CAN-057 OUT CLOSE
        [482].S.BITS2.31   // 90-CAN-057 OUT OPEN
        [483].S.BITS1.0   // 90-CAN-058 Enable
        [483].S.BITS1.1   // 90-CAN-058 Falla Resumen
        [483].S.BITS1.2   // 90-CAN-058 Conf Pos Abrir
        [483].S.BITS1.4   // 90-CAN-058 Conf Pos Cerrar
        [483].S.BITS1.29   // 90-CAN-058 Falla Abrir
        [483].S.BITS1.30   // 90-CAN-058 Falla Cerrar
        [483].S.BITS2.20   // 90-CAN-058 Reset Falla
        [483].S.BITS2.23   // 90-CAN-058 Test
        [483].S.BITS2.27   // 90-CAN-058 Cmd. Open
        [483].S.BITS2.30   // 90-CAN-058 OUT CLOSE
        [483].S.BITS2.31   // 90-CAN-058 OUT OPEN
        [484].S.BITS1.0   // 90-CAN-059 Enable
        [484].S.BITS1.1   // 90-CAN-059 Falla Resumen
        [484].S.BITS1.2   // 90-CAN-059 Conf Pos Abrir
        [484].S.BITS1.4   // 90-CAN-059 Conf Pos Cerrar
        [484].S.BITS1.29   // 90-CAN-059 Falla Abrir
        [484].S.BITS1.30   // 90-CAN-059 Falla Cerrar
        [484].S.BITS2.20   // 90-CAN-059 Reset Falla
        [484].S.BITS2.23   // 90-CAN-059 Test
        [484].S.BITS2.27   // 90-CAN-059 Cmd. Open
        [484].S.BITS2.30   // 90-CAN-059 OUT CLOSE
        [484].S.BITS2.31   // 90-CAN-059 OUT OPEN
        [485].S.BITS1.0   // 90-CAN-060 Enable
        [485].S.BITS1.1   // 90-CAN-060 Falla Resumen
        [485].S.BITS1.2   // 90-CAN-060 Conf Pos Abrir
        [485].S.BITS1.4   // 90-CAN-060 Conf Pos Cerrar
        [485].S.BITS1.26   // 90-TDC-020 FLL
        [485].S.BITS1.27   // 90-TDC-020 FV0
        [485].S.BITS1.28   // 90-TDC-020 FATO
        [485].S.BITS1.29   // 90-CAN-060 Falla Abrir
        [485].S.BITS1.30   // 90-CAN-060 Falla Cerrar
        [485].S.BITS2.20   // 90-CAN-060 Reset Falla
        [485].S.BITS2.23   // 90-CAN-060 Test
        [485].S.BITS2.27   // 90-CAN-060 Cmd. Open
        [485].S.BITS2.30   // 90-CAN-060 OUT CLOSE
        [485].S.BITS2.31   // 90-CAN-060 OUT OPEN
        [486].S.BITS1.0   // 90-CAN-061 Enable
        [486].S.BITS1.1   // 90-CAN-061 Falla Resumen
        [486].S.BITS1.2   // 90-CAN-061 Conf Pos Abrir
        [486].S.BITS1.4   // 90-CAN-061 Conf Pos Cerrar
        [486].S.BITS1.29   // 90-CAN-061 Falla Abrir
        [486].S.BITS1.30   // 90-CAN-061 Falla Cerrar
        [486].S.BITS2.20   // 90-CAN-061 Reset Falla
        [486].S.BITS2.23   // 90-CAN-061 Test
        [486].S.BITS2.27   // 90-CAN-061 Cmd. Open
        [486].S.BITS2.30   // 90-CAN-061 OUT CLOSE
        [486].S.BITS2.31   // 90-CAN-061 OUT OPEN
        [487].S.BITS1.0   // 90-CAN-064 Enable
        [487].S.BITS1.1   // 90-CAN-064 Falla Resumen
        [487].S.BITS1.2   // 90-CAN-064 Conf Pos Abrir
        [487].S.BITS1.4   // 90-CAN-064 Conf Pos Cerrar
        [487].S.BITS1.29   // 90-CAN-064 Falla Abrir
        [487].S.BITS1.30   // 90-CAN-064 Falla Cerrar
        [487].S.BITS2.20   // 90-CAN-064 Reset Falla
        [487].S.BITS2.23   // 90-CAN-064 Test
        [487].S.BITS2.27   // 90-CAN-064 Cmd. Open
        [487].S.BITS2.30   // 90-CAN-064 OUT CLOSE
        [487].S.BITS2.31   // 90-CAN-064 OUT OPEN
        [488].S.BITS1.0   // 90-TDC-016 Enable
        [488].S.BITS1.1   // 90-TDC-016 Falla Resumen
        [488].S.BITS1.2   // 90-TDC-016 Conf. Marcha
        [488].S.BITS1.4   // 90-TDC-016 Cmd. Automatico
        [488].S.BITS1.26   // 90-TDC-016 FLL
        [488].S.BITS1.27   // 90-TDC-016 FV0
        [488].S.BITS1.28   // 90-TDC-016 FATO
        [488].S.BITS1.29   // 90-CAN-065 Falla Abrir
        [488].S.BITS1.30   // 90-TDC-016 Falla Partida
        [488].S.BITS2.20   // 90-TDC-016 Reset Falla
        [488].S.BITS2.23   // 90-TDC-016 Test
        [488].S.BITS2.27   // 90-TDC-016 Cmd. Marcha
        [488].S.BITS2.30   // 90-TDC-016 OUT MARCHA
        [488].S.BITS2.31   // 90-CAN-065 OUT OPEN
        [489].S.BITS1.0   // 90-CAN-068 Enable
        [489].S.BITS1.1   // 90-CAN-068 Falla Resumen
        [489].S.BITS1.2   // 90-CAN-068 Conf Pos Abrir
        [489].S.BITS1.4   // 90-CAN-068 Conf Pos Cerrar
        [489].S.BITS1.29   // 90-CAN-068 Falla Abrir
        [489].S.BITS1.30   // 90-CAN-068 Falla Cerrar
        [489].S.BITS2.20   // 90-CAN-068 Reset Falla
        [489].S.BITS2.23   // 90-CAN-068 Test
        [489].S.BITS2.27   // 90-CAN-068 Cmd. Open
        [489].S.BITS2.30   // 90-CAN-068 OUT CLOSE
        [489].S.BITS2.31   // 90-CAN-068 OUT OPEN
        [490].S.BITS1.0   // 90-CAN-070 Enable
        [490].S.BITS1.1   // 90-CAN-070 Falla Resumen
        [490].S.BITS1.2   // 90-CAN-070 Conf Pos Abrir
        [490].S.BITS1.4   // 90-CAN-070 Conf Pos Cerrar
        [490].S.BITS1.29   // 90-CAN-070 Falla Abrir
        [490].S.BITS1.30   // 90-CAN-070 Falla Cerrar
        [490].S.BITS2.20   // 90-CAN-070 Reset Falla
        [490].S.BITS2.23   // 90-CAN-070 Test
        [490].S.BITS2.27   // 90-CAN-070 Cmd. Open
        [490].S.BITS2.30   // 90-CAN-070 OUT CLOSE
        [490].S.BITS2.31   // 90-CAN-070 OUT OPEN
        [491].S.BITS1.0   // 90-CAN-071 Enable
        [491].S.BITS1.1   // 90-CAN-071 Falla Resumen
        [491].S.BITS1.2   // 90-CAN-071 Conf Pos Abrir
        [491].S.BITS1.4   // 90-CAN-071 Conf Pos Cerrar
        [491].S.BITS1.29   // 90-CAN-071 Falla Abrir
        [491].S.BITS1.30   // 90-CAN-071 Falla Cerrar
        [491].S.BITS2.20   // 90-CAN-071 Reset Falla
        [491].S.BITS2.23   // 90-CAN-071 Test
        [491].S.BITS2.27   // 90-CAN-071 Cmd. Open
        [491].S.BITS2.30   // 90-CAN-071 OUT CLOSE
        [491].S.BITS2.31   // 90-CAN-071 OUT OPEN
        [492].S.BITS1.0   // 90-CAN-072 Enable
        [492].S.BITS1.1   // 90-CAN-072 Falla Resumen
        [492].S.BITS1.2   // 90-CAN-072 Conf Pos Abrir
        [492].S.BITS1.4   // 90-CAN-072 Conf Pos Cerrar
        [492].S.BITS1.29   // 90-CAN-072 Falla Abrir
        [492].S.BITS1.30   // 90-CAN-072 Falla Cerrar
        [492].S.BITS2.20   // 90-CAN-072 Reset Falla
        [492].S.BITS2.23   // 90-CAN-072 Test
        [492].S.BITS2.27   // 90-CAN-072 Cmd. Open
        [492].S.BITS2.30   // 90-CAN-072 OUT CLOSE
        [492].S.BITS2.31   // 90-CAN-072 OUT OPEN
        [236].S.BITS1.30   // 100-CAN-025 Falla Cerrar
        [607].S.BITS1.10   // 120-CAN-044 Conf. Abierto
        [297].S.BITS1.0   // 100-TOL-003-1 Enable
        [297].S.BITS2.23   // 100-TOL-003-1 Test
        [474].S.BITS1.8   // 110-TOR-002/2 Atollo
        [322].S.BITS2.31   // 100-MIX-001-M OUT MARCHA
        [608].S.BITS1.10   // 120-CAN-045 Conf. Abierto
        [494].S.BITS1.8   // 90-SIL-041 LL
        [494].S.BITS1.10   // 110-CAN-009/3 Conf. Abierto
        [309].S.BITS2.31   // XY-6100 OUT MARCHA
        [385].S.BITS2.23   // 110-ENF-001/1-2 Test
        [475].S.BITS1.8   // 110-TOR-003/2 Atollo
        [365].S.BITS2.31   // 110-CAN-010/1 OUT MARCHA
        [612].S.BITS1.10   // 120-CAN-055 Conf. Abierto
        [495].S.BITS1.29   // 90-CAN-075 Falla Abrir
        [405].S.BITS2.23   // 9-CON-667 Test
        [445].S.BITS2.23   // 9-CON-707 Test
        [496].S.BITS1.0   // 90-CAN-076 Enable
        [496].S.BITS1.1   // 90-CAN-076 Falla Resumen
        [496].S.BITS1.2   // 90-CAN-076 Conf Pos Abrir
        [496].S.BITS1.4   // 90-CAN-076 Conf Pos Cerrar
        [496].S.BITS1.29   // 90-CAN-076 Falla Abrir
        [496].S.BITS1.30   // 90-CAN-076 Falla Cerrar
        [496].S.BITS2.20   // 90-CAN-076 Reset Falla
        [496].S.BITS2.23   // 90-CAN-076 Test
        [496].S.BITS2.27   // 90-CAN-076 Cmd. Open
        [496].S.BITS2.30   // 90-CAN-076 OUT CLOSE
        [496].S.BITS2.31   // 90-CAN-076 OUT OPEN
        [497].S.BITS1.8   // 90-SIL-044 LL
        [498].S.BITS1.0   // 90-TDC-019 Enable
        [498].S.BITS1.1   // 90-TDC-019 Falla Resumen
        [498].S.BITS1.2   // 90-TDC-019 Conf. Marcha
        [498].S.BITS1.4   // 90-TDC-019 Cmd. Automatico
        [498].S.BITS1.8   // 90-SIL-045 LL
        [498].S.BITS1.9   // 90-SIL-045 LM
        [498].S.BITS1.10   // 90-SIL-045 LH
        [498].S.BITS1.26   // 90-TDC-019 FLL
        [498].S.BITS1.27   // 90-TDC-019 FV0
        [498].S.BITS1.28   // 90-TDC-019 FATO
        [498].S.BITS1.30   // 90-TDC-019 Falla Partida
        [498].S.BITS2.20   // 90-TDC-019 Reset Falla
        [498].S.BITS2.23   // 90-TDC-019 Test
        [498].S.BITS2.27   // 90-TDC-019 Cmd. Marcha
        [498].S.BITS2.30   // 90-TDC-019 OUT MARCHA
        [499].S.BITS1.0   // 90-CAN-048 Enable
        [499].S.BITS1.1   // 90-CAN-048 Falla Resumen
        [499].S.BITS1.2   // 90-CAN-048 Conf Pos Abrir
        [499].S.BITS1.4   // 90-CAN-048 Conf Pos Cerrar
        [499].S.BITS1.29   // 90-CAN-048 Falla Abrir
        [499].S.BITS1.30   // 90-CAN-048 Falla Cerrar
        [499].S.BITS2.20   // 90-CAN-048 Reset Falla
        [499].S.BITS2.23   // 90-CAN-048 Test
        [499].S.BITS2.27   // 90-CAN-048 Cmd. Open
        [499].S.BITS2.30   // 90-CAN-048 OUT CLOSE
        [499].S.BITS2.31   // 90-CAN-048 OUT OPEN
        [370].S.BITS2.31   // 110-TOR-001/1 OUT MARCHA
        [613].S.BITS1.10   // 120-CAN-056 Conf. Abierto
        [500].S.BITS1.29   // 90-CAN-049 Falla Abrir
        [465].S.BITS2.23   // 9-CON-727 Test
        [515].S.BITS2.23   // 110-ENF-001/3-2 Test
        [501].S.BITS1.0   // 90-CAN-050 Enable
        [501].S.BITS1.1   // 90-CAN-050 Falla Resumen
        [501].S.BITS1.2   // 90-CAN-050 Conf Pos Abrir
        [501].S.BITS1.4   // 90-CAN-050 Conf Pos Cerrar
        [501].S.BITS1.8   // 90-SIL-048 LL
        [501].S.BITS1.9   // 90-SIL-048 LM
        [501].S.BITS1.10   // 90-SIL-048 LH
        [501].S.BITS1.29   // 90-CAN-050 Falla Abrir
        [501].S.BITS1.30   // 90-CAN-050 Falla Cerrar
        [501].S.BITS2.20   // 90-CAN-050 Reset Falla
        [501].S.BITS2.23   // 90-CAN-050 Test
        [501].S.BITS2.27   // 90-CAN-050 Cmd. Open
        [501].S.BITS2.30   // 90-CAN-050 OUT CLOSE
        [501].S.BITS2.31   // 90-CAN-050 OUT OPEN
        [372].S.BITS2.31   // 110-ACD-001/1 OUT MARCHA
        [614].S.BITS1.10   // 120-CAN-057 Conf. Abierto
        [502].S.BITS1.29   // 90-CAN-051 Falla Abrir
        [535].S.BITS2.23   // 110-ENF-002/3-2 Test
        [560].S.BITS1.1   // CV-11 Falla Resumen
        [239].S.BITS1.8   // 100-MMA-001 Atollo
        [373].S.BITS2.31   // 110-EXP-001/1 OUT MARCHA
        [503].S.BITS1.2   // 110-EXP-001/3 Conf. Marcha
        [146].S.BITS1.10   // 100-TDC-004 Velocidad Cero
        [503].S.BITS1.29   // 90-.CAN-052 Falla Abrir
        [374].S.BITS2.31   // 110-DES-001/1 OUT MARCHA
        [337].S.BITS1.9   // 110-VEN-003 Sobrecarga
        [342].S.BITS1.9   // 110-TDC-001 Sobrecarga
        [503].S.BITS2.31   // 110-EXP-001/3 OUT MARCHA
        [504].S.BITS1.10   // 110-DES-001/3 Velocidad Cero
        [615].S.BITS1.10   // 120-CAN-058 Conf. Abierto
        [505].S.BITS1.10   // 110-CAE-001/3 Velocidad Cero
        [376].S.BITS2.31   // 110-PLT-001/1 OUT MARCHA
        [349].S.BITS1.9   // 8-TOL-712 LM
        [381].S.BITS2.31   // 110-ESC-001/1 OUT MARCHA
        [616].S.BITS1.10   // 120-CAN-059 Conf. Abierto
        [506].S.BITS1.29   // 90-CAN-063 Falla Abrir
        [560].S.BITS1.2   // CV-11 Conf Pos Abrir
        [560].S.BITS1.4   // CV-11 Conf Pos Cerrar
        [506].S.BITS2.31   // 110-PLT-001/3 OUT MARCHA
        [385].S.BITS2.31   // 110-ENF-001/1-2 OUT OPEN
        [617].S.BITS1.10   // 120-CAN-060 Conf. Abierto
        [507].S.BITS1.8   // 90-SIL-054 LL
        [507].S.BITS1.10   // 110-BIF-001/3 Conf. Pos Derecha
        [560].S.BITS1.30   // CV-11 Falla Cerrar
        [570].S.BITS1.1   // CV-12 Falla Resumen
        [476].S.BITS1.8   // 110-ELV-002/2 Atollo
        [508].S.BITS1.0   // 90-CAN-065 Enable
        [508].S.BITS1.1   // 90-CAN-065 Falla Resumen
        [508].S.BITS1.2   // 90-CAN-065 Conf Pos Abrir
        [508].S.BITS1.4   // 90-CAN-065 Conf Pos Cerrar
        [508].S.BITS1.8   // 90-SIL-055 LL
        [508].S.BITS1.9   // 90-SIL-055 LM
        [508].S.BITS1.10   // 90-SIL-055 LH
        [508].S.BITS1.29   // 90-CAN-065 Falla Abrir
        [508].S.BITS1.30   // 90-CAN-065 Falla Cerrar
        [508].S.BITS2.20   // 90-CAN-065 Reset Falla
        [508].S.BITS2.23   // 90-CAN-065 Test
        [508].S.BITS2.27   // 90-CAN-065 Cmd. Open
        [508].S.BITS2.30   // 90-CAN-065 OUT CLOSE
        [508].S.BITS2.31   // 90-CAN-065 OUT OPEN
        [509].S.BITS1.0   // 90-CAN-066 Enable
        [509].S.BITS1.1   // 90-CAN-066 Falla Resumen
        [509].S.BITS1.2   // 90-CAN-066 Conf Pos Abrir
        [509].S.BITS1.4   // 90-CAN-066 Conf Pos Cerrar
        [509].S.BITS1.8   // 90-SIL-056 LL
        [509].S.BITS1.9   // 90-SIL-056 LM
        [509].S.BITS1.10   // 90-SIL-056 LH
        [509].S.BITS1.29   // 90-CAN-066 Falla Abrir
        [509].S.BITS1.30   // 90-CAN-066 Falla Cerrar
        [509].S.BITS2.20   // 90-CAN-066 Reset Falla
        [509].S.BITS2.23   // 90-CAN-066 Test
        [509].S.BITS2.27   // 90-CAN-066 Cmd. Open
        [509].S.BITS2.30   // 90-CAN-066 OUT CLOSE
        [509].S.BITS2.31   // 90-CAN-066 OUT OPEN
        [510].S.BITS1.0   // 90-CAN-067 Enable
        [510].S.BITS1.1   // 90-CAN-067 Falla Resumen
        [510].S.BITS1.2   // 90-CAN-067 Conf Pos Abrir
        [510].S.BITS1.4   // 90-CAN-067 Conf Pos Cerrar
        [510].S.BITS1.29   // 90-CAN-067 Falla Abrir
        [510].S.BITS1.30   // 90-CAN-067 Falla Cerrar
        [510].S.BITS2.20   // 90-CAN-067 Reset Falla
        [510].S.BITS2.23   // 90-CAN-067 Test
        [510].S.BITS2.27   // 90-CAN-067 Cmd. Open
        [510].S.BITS2.30   // 90-CAN-067 OUT CLOSE
        [510].S.BITS2.31   // 90-CAN-067 OUT OPEN
        [512].S.BITS1.7   // 90-SIL-012 LLL
        [513].S.BITS1.7   // 90-SIL-011 LLL
        [514].S.BITS1.7   // 90-SIL-010 LLL
        [515].S.BITS1.7   // 90-SIL-009 LLL
        [515].S.BITS1.8   // 90-SIL-009 LL
        [515].S.BITS1.9   // 90-SIL-009 LM
        [515].S.BITS1.10   // 90-SIL-009 LH
        [516].S.BITS1.7   // 90-SIL-008 LLL
        [517].S.BITS1.7   // 90-SIL-007 LLL
        [518].S.BITS1.7   // 90-SIL-067 LLL
        [518].S.BITS1.8   // 90-SIL-067 LL
        [518].S.BITS1.9   // 90-SIL-067 LM
        [518].S.BITS1.10   // 90-SIL-067 LH
        [519].S.BITS1.7   // 90-SIL-068 LLL
        [520].S.BITS1.7   // 90-SIL-069 LLL
        [521].S.BITS1.7   // 90-SIL-70 LLL
        [522].S.BITS1.7   // 90-SIL-063 LLL
        [522].S.BITS1.8   // 90-SIL-063 LL
        [522].S.BITS1.9   // 90-SIL-063 LM
        [522].S.BITS1.10   // 90-SIL-063 LH
        [523].S.BITS1.7   // 90-SIL-064 LLL
        [524].S.BITS1.7   // 90-SIL-065 LLL
        [525].S.BITS1.7   // 90-SIL-066 LLL
        [525].S.BITS1.8   // 90-SIL-066 LL
        [525].S.BITS1.9   // 90-SIL-066 LM
        [525].S.BITS1.10   // 90-SIL-066 LH
        [526].S.BITS1.7   // 90-SIL-057 LLL
        [526].S.BITS1.8   // 90-SIL-057 LL
        [526].S.BITS1.9   // 90-SIL-057 LM
        [526].S.BITS1.10   // 90-SIL-057 LH
        [527].S.BITS1.7   // 90-SIL-058 LLL
        [527].S.BITS1.8   // 90-SIL-058 LL
        [527].S.BITS1.9   // 90-SIL-058 LM
        [527].S.BITS1.10   // 90-SIL-058 LH
        [528].S.BITS1.7   // 90-SIL-059 LLL
        [528].S.BITS1.8   // 90-SIL-059 LL
        [528].S.BITS1.9   // 90-SIL-059 LM
        [528].S.BITS1.10   // 90-SIL-059 LH
        [529].S.BITS1.7   // 90-SIL-060 LLL
        [529].S.BITS1.8   // 90-SIL-060 LL
        [529].S.BITS1.9   // 90-SIL-060 LM
        [529].S.BITS1.10   // 90-SIL-060 LH
        [530].S.BITS1.7   // 90-SIL-061 LLL
        [530].S.BITS1.8   // 90-SIL-061 LL
        [530].S.BITS1.9   // 90-SIL-061 LM
        [530].S.BITS1.10   // 90-SIL-061 LH
        [531].S.BITS1.7   // 90-SIL-062 LLL
        [532].S.BITS1.7   // 90-SIL-041 LLL
        [533].S.BITS1.7   // 90-SIL-042 LLL
        [534].S.BITS1.7   // 90-SIL-043 LLL
        [535].S.BITS1.7   // 90-SIL-044 LLL
        [535].S.BITS1.8   // 90-SIL-044 LL
        [535].S.BITS1.9   // 90-SIL-044 LM
        [535].S.BITS1.10   // 90-SIL-044 LH
        [536].S.BITS1.7   // 90-SIL-045 LLL
        [537].S.BITS1.7   // 90-SIL-046 LLL
        [538].S.BITS1.7   // 90-SIL-047 LLL
        [538].S.BITS1.8   // 90-SIL-047 LL
        [538].S.BITS1.9   // 90-SIL-047 LM
        [538].S.BITS1.10   // 90-SIL-047 LH
        [539].S.BITS1.7   // 90-SIL-048 LLL
        [540].S.BITS1.7   // 90-SIL-049 LLL
        [541].S.BITS1.7   // 90-SIL-050 LLL
        [542].S.BITS1.7   // 90-SIL-051 LLL
        [542].S.BITS1.8   // 90-SIL-051 LL
        [542].S.BITS1.9   // 90-SIL-051 LM
        [542].S.BITS1.10   // 90-SIL-051 LH
        [543].S.BITS1.7   // 90-SIL-052 LLL
        [543].S.BITS1.8   // 90-SIL-052 LL
        [543].S.BITS1.9   // 90-SIL-052 LM
        [543].S.BITS1.10   // 90-SIL-052 LH
        [544].S.BITS1.7   // 90-SIL-053 LLL
        [545].S.BITS1.7   // 90-SIL-054 LLL
        [546].S.BITS1.7   // 90-SIL-055 LLL
        [547].S.BITS1.7   // 90-SIL-056 LLL
        [549].S.BITS1.7   // TOL_VIR_DESP-03 LLL
        [549].S.BITS1.8   // TOL_VIR_DESP-03 LL
        [549].S.BITS1.9   // TOL_VIR_DESP-03 LM
        [549].S.BITS1.10   // TOL_VIR_DESP-03 LH
        [550].S.BITS1.0   // CV-10 Enable
        [550].S.BITS1.1   // CV-10 Falla Resumen
        [550].S.BITS1.2   // CV-10 Conf Pos Abrir
        [550].S.BITS1.4   // CV-10 Conf Pos Cerrar
        [550].S.BITS1.29   // CV-10 Falla Abrir
        [550].S.BITS1.30   // CV-10 Falla Cerrar
        [550].S.BITS2.20   // CV-10 Reset Falla
        [550].S.BITS2.23   // CV-10 Test
        [550].S.BITS2.27   // CV-10 Cmd. Open
        [550].S.BITS2.30   // CV-10 OUT CLOSE
        [550].S.BITS2.31   // CV-10 OUT OPEN
        [551].S.BITS1.7   // TOL_VIR_DESP-04 LLL
        [560].S.BITS1.29   // CV-11 Falla Abrir
        [560].S.BITS2.20   // CV-11 Reset Falla
        [552].S.BITS1.0   // 110-TDC-004/1 Enable
        [552].S.BITS1.1   // 110-TDC-004/1 Falla Resumen
        [552].S.BITS1.2   // 110-TDC-004/1 Conf. Marcha
        [552].S.BITS1.4   // 110-TDC-004/1 Cmd. Automatico
        [552].S.BITS1.29   // COM-VIR-DESP-04 Falla Abrir
        [552].S.BITS1.30   // 110-TDC-004/1 Falla Partida
        [552].S.BITS2.20   // 110-TDC-004/1 Reset Falla
        [552].S.BITS2.23   // 110-TDC-004/1 Test
        [552].S.BITS2.27   // 110-TDC-004/1 Cmd. Marcha
        [552].S.BITS2.30   // 110-TDC-004/1 OUT MARCHA
        [552].S.BITS2.31   // 110-TDC-004/1 OUT MARCHA
        [553].S.BITS1.7   // TOL_VIR_DESP-05 LLL
        [553].S.BITS1.8   // TOL_VIR_DESP-05 LL
        [553].S.BITS1.9   // TOL_VIR_DESP-05 LM
        [553].S.BITS1.10   // TOL_VIR_DESP-05 LH
        [554].S.BITS1.0   // 110-ELV-001/1 Enable
        [554].S.BITS1.1   // 110-ELV-001/1 Falla Resumen
        [554].S.BITS1.2   // 110-ELV-001/1 Conf. Marcha
        [554].S.BITS1.4   // 110-ELV-001/1 Cmd. Automatico
        [554].S.BITS1.29   // COM-VIR-DESP-05 Falla Abrir
        [554].S.BITS1.30   // 110-ELV-001/1 Falla Partida
        [554].S.BITS2.20   // 110-ELV-001/1 Reset Falla
        [554].S.BITS2.23   // 110-ELV-001/1 Test
        [554].S.BITS2.27   // 110-ELV-001/1 Cmd. Marcha
        [554].S.BITS2.30   // 110-ELV-001/1 OUT MARCHA
        [554].S.BITS2.31   // 110-ELV-001/1 OUT MARCHA
        [555].S.BITS1.7   // TOL_VIR_DESP-05 LLL
        [570].S.BITS1.29   // CV-12 Falla Abrir
        [570].S.BITS2.20   // CV-12 Reset Falla
        [41].S.BITS2.31   // 90-CAN-012 OUT OPEN
        [556].S.BITS1.0   // 120-HAR-001 Enable
        [556].S.BITS1.1   // 120-HAR-001 Falla Resumen
        [556].S.BITS1.2   // 120-HAR-001 Conf. Marcha
        [556].S.BITS1.4   // 120-HAR-001 Cmd. Automatico
        [556].S.BITS1.29   // COM-VIR-DESP-05 Falla Abrir
        [556].S.BITS1.30   // 120-HAR-001 Falla Partida
        [556].S.BITS2.20   // 120-HAR-001 Reset Falla
        [556].S.BITS2.23   // 120-HAR-001 Test
        [556].S.BITS2.27   // 120-HAR-001 Cmd. Marcha
        [556].S.BITS2.30   // 120-HAR-001 OUT MARCHA
        [556].S.BITS2.31   // 120-HAR-001 OUT MARCHA
        [313].S.BITS2.39   // M1-TRI-095 Out Izquierda
        [446].S.BITS2.39   // 90-TRI-001 Out Izquierda
        [447].S.BITS2.39   // 90-TRI-002 Out Izquierda
        [293].S.BITS2.31   // 100-ELV-002 OUT MARCHA
        [383].S.BITS1.7   // Nivel alto alto
        [13].S.BITS1.26   // 90-TDC-001 FLL
        [13].S.BITS1.27   // 90-TDC-001 FV0
        [13].S.BITS1.28   // 90-TDC-001 FATO
        [13].S.BITS1.30   // 7-CON-1013 Falla Cerrar
        [13].S.BITS2.27   // 7-CON-1013 Cmd. Open
        [13].S.BITS2.30   // 7-CON-1013 OUT CLOSE
        [16].S.BITS2.31   // 90-CAN-003 OUT OPEN
        [17].S.BITS2.31   // 90-CAN-004 OUT OPEN
        [18].S.BITS1.26   // 90-TDC-002 FLL
        [18].S.BITS1.27   // 90-TDC-002 FV0
        [18].S.BITS1.28   // 90-TDC-002 FATO
        [19].S.BITS1.0   // 7-RED-1019 Enable
        [19].S.BITS1.1   // 7-RED-1019 Falla Resumen
        [19].S.BITS1.2   // 7-RED-1019 Conf. Marcha
        [19].S.BITS1.4   // 7-RED-1019 Cmd. Automatico
        [19].S.BITS1.29   // 90-CAN-006 Falla Abrir
        [19].S.BITS2.20   // 7-RED-1019 Reset Falla
        [19].S.BITS2.23   // 7-RED-1019 Test
        [19].S.BITS2.31   // 90-CAN-006 OUT OPEN
        [20].S.BITS1.0   // 7-RED-1020 Enable
        [20].S.BITS1.1   // 7-RED-1020 Falla Resumen
        [20].S.BITS1.2   // 7-RED-1020 Conf. Marcha
        [20].S.BITS1.4   // 7-RED-1020 Cmd. Automatico
        [20].S.BITS1.29   // 90-CAN-007 Falla Abrir
        [20].S.BITS2.20   // 7-RED-1020 Reset Falla
        [20].S.BITS2.23   // 7-RED-1020 Test
        [20].S.BITS2.31   // 90-CAN-007 OUT OPEN
        [21].S.BITS1.0   // 7-COM-1021 Enable
        [21].S.BITS1.1   // 7-COM-1021 Falla Resumen
        [21].S.BITS1.2   // 7-COM-1021 Conf Pos Abrir
        [21].S.BITS1.4   // 7-COM-1021 Conf Pos Cerrar
        [21].S.BITS1.29   // 7-COM-1021 Falla Abrir
        [21].S.BITS1.30   // 7-COM-1021 Falla Cerrar
        [21].S.BITS2.20   // 7-COM-1021 Reset Falla
        [21].S.BITS2.23   // 7-COM-1021 Test
        [21].S.BITS2.27   // 7-COM-1021 Cmd. Open
        [21].S.BITS2.30   // 7-COM-1021 OUT CLOSE
        [21].S.BITS2.31   // 7-COM-1021 OUT OPEN
        [22].S.BITS1.0   // 7-COM-1022 Enable
        [22].S.BITS1.1   // 7-COM-1022 Falla Resumen
        [22].S.BITS1.2   // 7-COM-1022 Conf Pos Abrir
        [22].S.BITS1.4   // 7-COM-1022 Conf Pos Cerrar
        [22].S.BITS1.29   // 7-COM-1022 Falla Abrir
        [22].S.BITS1.30   // 7-COM-1022 Falla Cerrar
        [22].S.BITS2.20   // 7-COM-1022 Reset Falla
        [22].S.BITS2.23   // 7-COM-1022 Test
        [22].S.BITS2.27   // 7-COM-1022 Cmd. Open
        [22].S.BITS2.30   // 7-COM-1022 OUT CLOSE
        [22].S.BITS2.31   // 7-COM-1022 OUT OPEN
        [23].S.BITS1.0   // 7-COM-1023 Enable
        [23].S.BITS1.1   // 7-COM-1023 Falla Resumen
        [23].S.BITS1.2   // 7-COM-1023 Conf Pos Abrir
        [23].S.BITS1.4   // 7-COM-1023 Conf Pos Cerrar
        [23].S.BITS1.29   // 7-COM-1023 Falla Abrir
        [23].S.BITS1.30   // 7-COM-1023 Falla Cerrar
        [23].S.BITS2.20   // 7-COM-1023 Reset Falla
        [23].S.BITS2.23   // 7-COM-1023 Test
        [23].S.BITS2.27   // 7-COM-1023 Cmd. Open
        [23].S.BITS2.30   // 7-COM-1023 OUT CLOSE
        [23].S.BITS2.31   // 7-COM-1023 OUT OPEN
        [24].S.BITS1.0   // 7-RED-1024 Enable
        [24].S.BITS1.1   // 7-RED-1024 Falla Resumen
        [24].S.BITS1.2   // 7-RED-1024 Conf. Marcha
